(* CoDeSys 2.3 export: CELA.EXP *)

(* Data type in EPT Lib/Achsen/BECKHOFF *)
TYPE enum_ecd_cmd :
	(
	NO_COMMAND := 0,
	ABORT,
	POWER_DISABLE,
	POWER_ENABLE,
	RESET,
	HOME,
	SET_POSITION,
	JOG_VORWAERTS,
	JOG_RUECKWAERTS,
	JOG_STOP,
	MOVE_ABSOLUTE,
	MOVE_ABSOLUTE_NEXT,
	MOVE_RELATIVE,
	MOVE_VELOCITY,
	MOVE_MODULO,
	MOVE_TOUCH_PROBE,
	STOP_AXIS,
	HALT_AXIS,
	GEAR_IN_SLAVE,
	GEAR_OUT_SLAVE,
	CAM_IN_SLAVE,
	CAM_OUT_SLAVE,
	CAM_SCALEING_SLAVE,
	SOE_WRITE_PARAM,
	SOE_READ_PARAM,
	ECCOESDO_WRITE_PARAM,
	ECCOESDO_READ_PARAM,
	WRITE_NC_PARAMETER,
	READ_NC_PARAMETER,
	WRITE_ADS_PARAMETER,
	READ_ADS_PARAMETER,
	WRITE_MOTION_POINT,
	READ_MOTION_POINT,
	READ_SLAVE_DYNAMICS,
	READ_CAMTABLE_CHAR

	);
END_TYPE

(* Data type in EPT Lib/Achsen/BECKHOFF *)
TYPE enum_ecd_typ :
	(
	LINEAR := 1,
	RUND,
	LINEAR_VIRTUELL,
	RUND_VIRTUELL,
	SERVOKLEMME7201
	);
END_TYPE

(* Data type in EPT Lib/Achsen/BECKHOFF *)
TYPE st_camscaleingoptions :
STRUCT
	st_scaleing_activation_mode			: MC_CamActivationMode;
	r_scaleing_activation_position			: LREAL;
	st_master_scaling_mode				: MC_CamScalingMode;
	st_slave_scaling_mode				: MC_CamScalingMode;
END_STRUCT
END_TYPE

(* Data type in EPT Lib/Achsen/BECKHOFF *)
TYPE struct_achse :
STRUCT
	st_ctrl		: struct_ctrl;
	st_config		: struct_ecd_config;
	st_visu		: struct_ecd_visu;
END_STRUCT
END_TYPE

(* Data type in EPT Lib/Achsen/BECKHOFF *)
TYPE struct_ads_info :
STRUCT
	s_net_id 								: T_AmsNetId := '';
	st_symbol_info						: SYMINFOSTRUCT;
	dw_zieladresse_ads_read				: DWORD := 16#0000;
	dw_quelladresse_ads_write				: DWORD := 16#0000;
END_STRUCT
END_TYPE

(* Data type in EPT Lib/Achsen/BECKHOFF *)
TYPE struct_eccoe_sdo :
STRUCT
	s_ec_slave_net_id 		: T_AmsNetId := '';
	ui16_slave_addr 			: UINT := 0; (* Address of the slave device.*)
	i8_sub_index 				: BYTE := 0; (* CANopen Sdo subindex.*)
	w_index 					: WORD := 16#00; (* CANopen Sdo index.*)
	dw_p_source_buffer 		: DWORD := 16#0000; (* Contains the address of the buffer containing the data to be send. *)
	dw_p_destination_buffer	: DWORD := 16#0000; (* Contains the address of the buffer for the received data. *)
	ui32_buffer_length 			: UDINT := 0; (* Contains the max. number of bytes to be received. *)
	ui32_value 				: UDINT := 0; (* variable to be written to the CoE Object *)
	ui16_value 				: UINT := 0; (* variable to be written to the CoE Object *)
	byte_value 				: BYTE := 16#00; (* variable to be written to the CoE Object *)
	bool_value 				: BOOL := FALSE; (* variable to be written to the CoE Object *)
END_STRUCT
END_TYPE

(* Data type in EPT Lib/Achsen/BECKHOFF *)
TYPE struct_ecd_cmd :
STRUCT
	b_job_fehler 		: BOOL := FALSE;
	enu_cmd			: enum_ecd_cmd;
	meldungen		: struct_ecd_cmd_meldungen;
END_STRUCT
END_TYPE

(* Data type in EPT Lib/Achsen/BECKHOFF *)
TYPE struct_ecd_cmd_meldungen :
STRUCT
	sm_power_enable					: BOOL := FALSE;
	sm_power_disable				: BOOL := FALSE;
	sm_reset							: BOOL := FALSE;
	sm_home						: BOOL := FALSE;
	sm_setposition					: BOOL := FALSE;
	sm_jog_vorwaerts					: BOOL := FALSE;
	sm_jog_rueckwaerts				: BOOL := FALSE;
	sm_move_absolute				: BOOL := FALSE;
	sm_move_relative					: BOOL := FALSE;
	sm_move_velocity				: BOOL := FALSE;
	sm_move_modulo					: BOOL := FALSE;
	sm_stop_axis						: BOOL := FALSE;
	sm_halt_axis						: BOOL := FALSE;
	sm_gear_in_slave					: BOOL := FALSE;
	sm_gear_out_slave				: BOOL := FALSE;
	sm_cam_in_slave					: BOOL := FALSE;
	sm_cam_out_slave				: BOOL := FALSE;
	sm_cam_scaleing_slave			: BOOL := FALSE;
	sm_motion_command_timeout		: BOOL := FALSE;
	sm_camgear_command_timeout	: BOOL := FALSE;
	sm_achse_nicht_referenziert		: BOOL := FALSE;
	sm_limit_positiv_erreicht			: BOOL := FALSE;
	sm_limit_negativ_erreicht			: BOOL := FALSE;
	sm_write_soe_parameter			: BOOL := FALSE;
	sm_read_soe_parameter			: BOOL := FALSE;
	sm_write_nc_parameter			: BOOL := FALSE;
	sm_read_nc_parameter			: BOOL := FALSE;
	sm_write_motion_funktion_point		: BOOL := FALSE;
	sm_read_motion_funktion_point		: BOOL := FALSE;
	sm_read_camtable_slave_dynamics	: BOOL := FALSE;
	sm_read_camtable_charakteristik	: BOOL := FALSE;
	sm_write_ads_parameter			: BOOL := FALSE;
	sm_read_ads_parameter			: BOOL := FALSE;
	sm_ec_coe_sdo_write_ex			: BOOL := FALSE;
	sm_ec_coe_sdo_read_ex			: BOOL := FALSE;
	sm_touch_probe_defect			: BOOL := FALSE;
	sm_touch_probe_err				: BOOL := FALSE;
END_STRUCT
END_TYPE

(* Data type in EPT Lib/Achsen/BECKHOFF *)
TYPE struct_ecd_config :
STRUCT
	s_instanz_name					: STRING(48) := '';
	s_beschreibung					: STRING(32) := '';
	i16_meld_startindex				: INT;
	ui16_ethercat_adr					: UINT := 0;
	ui16_ethercat_slave_id				: UINT := 0;

	i16_achs_nr						: INT := 0;
	i16_modul_nr						: INT := 0;

	b_refsensor_vorhanden			: BOOL := FALSE;
	b_limitsensor_positiv_vorhanden	: BOOL := FALSE;
	b_limitsensor_negativ_vorhanden	: BOOL := FALSE;

	r_getriebefaktor					: LREAL := 0.0;
	ui16_bipolar_torque_limit			: UINT := 1000;
	i16_achstyp						: enum_ecd_typ;

	b_config_fertig					: BOOL := FALSE;
END_STRUCT
END_TYPE

(* Data type in EPT Lib/Achsen/BECKHOFF *)
TYPE struct_ecd_fehler :
STRUCT
	b_sammel				: BOOL := FALSE;
	b_job_fehler 				: BOOL := FALSE;
	b_achsfehler 				: BOOL := FALSE;
	b_devicefehler 			: BOOL := FALSE;
	b_limit_positiv_erreicht 		: BOOL := FALSE;
	b_limit_negativ_erreicht	: BOOL := FALSE;
END_STRUCT
END_TYPE

(* Data type in EPT Lib/Achsen/BECKHOFF *)
TYPE struct_ecd_geschwindigkeiten :
STRUCT
	lr_maximalgeschwindigkeit	: LREAL := 0.0;
	lr_beschleunigung 		: LREAL := 0.0;
	lr_verzoegerung	 		: LREAL := 0.0;
	lr_ruck			 		: LREAL := 0.0;

	lr_auto_max				: LREAL := 0.0;
	lr_auto_min				: LREAL := 0.0;
	lr_jog					: LREAL := 0.0;
END_STRUCT
END_TYPE

(* Data type in EPT Lib/Achsen/BECKHOFF *)
TYPE struct_ecd_meldungen :
STRUCT
	b_achsfehler					: BOOL := FALSE;
	b_devicefehler				: BOOL := FALSE;
	b_achse_nicht_bb				: BOOL := FALSE;
	b_achse_nicht_referenziert		: BOOL := FALSE;
	b_keine_verfahrfreigabe		: BOOL := FALSE;
	b_achse_nicht_auf_startpos		: BOOL := FALSE;
	b_ende_skalierungs_nocke		: BOOL := FALSE;
	b_ende_camming_nocke		: BOOL := FALSE;
	b_skalierung_noch_aktiv		: BOOL := FALSE;
END_STRUCT
END_TYPE

(* Data type in EPT Lib/Achsen/BECKHOFF *)
TYPE struct_ecd_positionen :
STRUCT
	r_soll		 			: LREAL := 0.0;
	r_referenz				: LREAL := 0.0;
	lr_ibn_pos_start			: LREAL := 0.0;
	lr_ibn_pos_ziel			: LREAL := 0.0;
END_STRUCT
END_TYPE

(* Data type in EPT Lib/Achsen/BECKHOFF *)
TYPE struct_ecd_visu :
STRUCT
	b_nullpunkt_setzen				: BOOL := FALSE;
	b_tippen_vorwaerts				: BOOL := FALSE;
	b_tippen_rueckwaerts				: BOOL := FALSE;
	b_achse_lueften					: BOOL := FALSE;
	b_achse_regeln					: BOOL := FALSE;
	b_bandeinzug_referenzieren		: BOOL := FALSE;
	i32_geschwindigkeit_soll			: DINT := 0;
	i32_geschwindigkeit_ist			: DINT := 0;
	i32_position_ist					: DINT := 0;
	lr_geschwindigkeit_soll				: LREAL := 0.0;
	lr_geschwindigkeit_ist				: LREAL := 0.0;
	lr_position_ist						: LREAL := 0.0;
	b_winkel_vor_ot_uebernehmen		: BOOL := FALSE;
	b_winkel_nach_ot_uebernehmen	: BOOL := FALSE;
	b_winkeloffset_uebernehmen		: BOOL := FALSE;
	b_einschalten						: BOOL := FALSE;
	b_ausschalten					: BOOL := FALSE;
	b_motor_dreht					: BOOL := FALSE;
	b_taste_vorgabegeschwindigkeit	: BOOL := FALSE;
	b_taste_plus						: BOOL := FALSE;
	b_taste_plusplus					: BOOL := FALSE;
	b_taste_minus					: BOOL := FALSE;
	b_taste_minusminus				: BOOL := FALSE;
	st_zyl							: struct_zylinder_visu;
END_STRUCT
END_TYPE

(* Data type in EPT Lib/Achsen/BECKHOFF *)
TYPE struct_nc_scaling_parameter :
STRUCT
	lr_ref_velo					: LREAL := 0.0;
	lr_max_velo					: LREAL := 0.0;
	lr_manual_velo_fast			: LREAL := 0.0;
	lr_manual_velo_slow			: LREAL := 0.0;
	lr_calibration_velo_forward		: LREAL := 0.0;
	lr_calibration_velo_backward	: LREAL := 0.0;
	lr_acceleration				: LREAL := 0.0;
	lr_deceleration				: LREAL := 0.0;
	lr_jerk						: LREAL := 0.0;
	lr_scaling_factor				: LREAL := 0.0;
END_STRUCT
END_TYPE

(* Data type in EPT Lib/Allgemeine Kontrollstrukturen Objekte *)
TYPE enum_step_nr :
	(
	INIT_OBJ := 0,
	INIT := 10,
	BEREIT := 100,
	FEHLER := 1000,
	STOP := 1100,
	STILLSTAND := 1200,
	HALT := 1300,
	HANDRAD := 2000,
	MOTORBREMSE_AUF :=2100,
	MOTORBREMSE_ZU := 2200,
	LUEFTEN := 2300,
	REGELN := 2400,
	NULLPUNKT_SETZEN := 2500,
	INBETRIEBNAHME := 5000,
	(* Zylinder *)
	ZYL_INIT := 3000,
	GESTOPPT := 3010,
	EINGEFAHREN := 3020,
	BEWEGUNG_AUSFAHREN := 3030,
	AUSGEFAHREN := 3040,
	BEWEGUNG_EINFAHREN := 3050,
	MITTEGEFAHREN := 3060,
	BEWEGUNG_MITTE := 3070,
	LUFTLOS := 3080,
	ZYL_FEHLER := 3090,
	DIREKT_EINFAHREN := 3100,
	DIREKT_AUSFAHREN := 3110
	);
END_TYPE

(* Data type in EPT Lib/Allgemeine Kontrollstrukturen Objekte *)
TYPE struct_config :
STRUCT
	str_instanz_name					: STRING(48) := '';
	str_beschreibung					: STRING(32) := '';
	b_station_aktiv					: BOOL := FALSE;
	b_station_in_simulation				: BOOL := FALSE;
	i16_meld_startindex				: INT := 0;
	b_config_fertig					: BOOL := FALSE;
END_STRUCT
END_TYPE

(* Data type in EPT Lib/Allgemeine Kontrollstrukturen Objekte *)
TYPE struct_ctrl :
STRUCT
	in		: struct_ctrl_in;
	out		: struct_ctrl_out;
END_STRUCT
END_TYPE

(* Data type in EPT Lib/Allgemeine Kontrollstrukturen Objekte *)
TYPE struct_ctrl_in :
STRUCT
	b_quitt						: BOOL := FALSE;
	b_stop 						: BOOL := FALSE;
         b_halt		  	 			: BOOL := FALSE;
         b_definierter_halt  	 			: BOOL := FALSE;
	b_init 						: BOOL := FALSE;
	b_init_2 						: BOOL := FALSE;
         b_preinit                				: BOOL := FALSE;
	b_start						: BOOL := FALSE;
	b_start_2						: BOOL := FALSE;
	b_gutteil_produziert 			: BOOL := FALSE;
	b_schlechtteil_produziert 		: BOOL := FALSE;
	b_start_lesen					: BOOL := FALSE;
	b_start_schreiben				: BOOL := FALSE;
	b_schutzhaube_ab			: BOOL := FALSE;
	b_schutzhaube_auf			: BOOL := FALSE;
	b_nachtabschaltung			: BOOL := FALSE;
	b_gehe_step_ibn				: BOOL := FALSE;
	b_ibn_start					: BOOL := FALSE;
	b_freigabe					: BOOL := FALSE;
	b_bremse_auf				: BOOL := FALSE;
	b_bremse_zu					: BOOL := FALSE;
	b_home						: BOOL := FALSE;
	b_ausfaedeln_servo			: BOOL := FALSE;
	b_einfaedeln_servo			: BOOL := FALSE;
	b_startpos					: BOOL := FALSE;
END_STRUCT
END_TYPE

(* Data type in EPT Lib/Allgemeine Kontrollstrukturen Objekte *)
TYPE struct_ctrl_out :
STRUCT
	b_bereit 						: BOOL := FALSE;
	b_bereit_2					: BOOL := FALSE;
         b_prebereit               			: BOOL := FALSE;
	b_fehler 						: BOOL := FALSE;
	b_fertig						: BOOL := FALSE;
	b_fertig_2					: BOOL := FALSE;
	b_bandende					: BOOL := FALSE;
	b_kontroller_start				: BOOL := FALSE;
	b_gestoppt					: BOOL := FALSE;
	b_angehalten					: BOOL := FALSE;
	b_haube_oeffnen				: BOOL := FALSE;
	b_nachtabschaltung			: BOOL := FALSE;
	b_einzelfertigung				: BOOL := FALSE;
	b_busy						: BOOL := FALSE;
	b_bremse_geschlossen		: BOOL := FALSE;
	b_bremse_geoeffnet			: BOOL := FALSE;
	b_ausgefaedelt_servo			: BOOL := FALSE;
	b_servo_auf_einfaedelpos		: BOOL := FALSE;
END_STRUCT
END_TYPE

(* Data type in EPT Lib/Allgemeine Kontrollstrukturen Objekte *)
TYPE struct_objekt :
STRUCT
	st_config		: struct_config;
	st_ctrl		: struct_ctrl;
	st_visu		: struct_visu;
END_STRUCT
END_TYPE

(* Data type in EPT Lib/Analogkarte *)
TYPE struct_analog_in :
STRUCT
	e_b_status_underrange		: BOOL := FALSE;
	e_b_status_overrange			: BOOL := FALSE;
	e_by_status_limit1				: BYTE := 2#0;
	e_by_status_limit2				: BYTE := 2#0;
	e_b_status_error				: BOOL := FALSE;
	e_i16_value					: INT := 0;
END_STRUCT
END_TYPE

(* Data type in EPT Lib/Analogkarte *)
TYPE struct_analogin :
STRUCT
	fb			: ST_AnalogIn;
	st_ctrl		: struct_ctrl;
END_STRUCT
END_TYPE

(* Data type in EPT Lib/Analogkarte *)
TYPE struct_analogout :
STRUCT
	fb			: ST_AnalogOut;
	st_ctrl		: struct_ctrl;
END_STRUCT
END_TYPE

(* Data type in EPT Lib/Betriebsarten *)
TYPE enum_betriebsarten :
	(KEINE := 0,
	AUTO,
	TIPPEN,
	DUMMY,
	PSEUDO,
	HAND);
END_TYPE

(* Data type in EPT Lib/Betriebsarten *)
TYPE struct_betriebsarten :
STRUCT
	st_config					: struct_config;
	st_ctrl					: struct_ctrl;
END_STRUCT
END_TYPE

(* Data type in EPT Lib/CamEditor *)
TYPE enum_auftrag_cameditor :
	(
	MFP_KEIN_AUFTRAG := 0,
	MFP_LESEN,
	MFP_SCHREIBEN
	);
END_TYPE

(* Data type in EPT Lib/CamEditor *)
TYPE struct_cam_editor :
STRUCT
	fb					: ST_Kurvenscheibeneditor;
	st_config				: struct_config;
	st_ctrl				: struct_ctrl;
END_STRUCT
END_TYPE

(* Data type in EPT Lib/CamEditor *)
TYPE struct_cameditor_meldungen :
STRUCT
	schreibe_mfp 							: BOOL := FALSE;
	lese_mfp									: BOOL := FALSE;
	schreibe_camtable						: BOOL := FALSE;
	lese_camtable							: BOOL := FALSE;
	berechne_konstantfahrphase				: BOOL := FALSE;
	berechne_max_master_geschwindigkeit		: BOOL := FALSE;
	lesen_werte_mf_tab						: BOOL := FALSE;
	fehler_cam_in								: BOOL := FALSE;
END_STRUCT
END_TYPE

(* Data type in EPT Lib/CamEditor *)
TYPE struct_camtable_maker :
STRUCT
	fb					: ST_Camtable_Maker;
	st_config			: struct_config;
	st_ctrl				: struct_ctrl;
END_STRUCT
END_TYPE

(* Data type in EPT Lib/CamEditor *)
TYPE struct_db_motionfunctionpoint :
STRUCT
	    PointIndex        		: MC_MotionFunctionPoint_ID;
	    FunctionType    		: MC_MotionFunctionType;
	    PointType        		: MC_MotionPointType;
	    MasterPos        		: LREAL; (* X *)
	    SlavePos          		: LREAL; (* Y *)
END_STRUCT
END_TYPE

(* Data type in EPT Lib/CamEditor *)
TYPE struct_mf_editor :
STRUCT
	fb					: ST_MFCalcConstPhase;
	st_config				: struct_config;
	st_ctrl				: struct_ctrl;
END_STRUCT
END_TYPE

(* Data type in EPT Lib/Diagnose *)
TYPE struct_ecat_klemmen_diagnose :
STRUCT
	WcState			: BOOL := 2#0;		(* 1 = Data invalid *)
	ECatState		: UINT := 0;		(* 0x08 = OP-State *)
END_STRUCT
END_TYPE

(* Data type in EPT Lib/Nockenschaltwerk/NSW_INT *)
TYPE struct_nocken_int :
STRUCT
	i16_track_no 				: INT := 0;
	b_camvalid 				: BOOL := FALSE;
	b_eff_direction_pos 		: BOOL := FALSE;
	b_eff_direction_neg 		: BOOL := FALSE;
	b_nockenzustand 			: BOOL := FALSE;
	i16_cam_begin 			: INT := 0;
	i16_cam_end 				: INT := 0;
	t_vorsteuerzeit			: TIME := t#0ms;
	i16_vorsteuerpos			: INT := 0;
END_STRUCT
END_TYPE

(* Data type in EPT Lib/Nockenschaltwerk/NSW_INT *)
TYPE struct_nockenschaltwerk_int :
STRUCT
	fb					: ST_Nockenschaltwerk_int;
	st_config				: struct_config;
	arr_nocken			: ARRAY [0..MAX_NOCKENGERUEST] OF struct_nocken_int;
	arr_spur				: ARRAY [0..MAX_NOCKENGERUEST] OF BOOL;
END_STRUCT
END_TYPE

(* Data type in EPT Lib/Nockenschaltwerk/NSW_LREAL *)
TYPE struct_nocken_lreal :
STRUCT
	i16_track_no 				: INT := 0;
	b_camvalid 				: BOOL := FALSE;
	b_eff_direction_pos 		: BOOL := FALSE;
	b_eff_direction_neg 		: BOOL := FALSE;
	b_nockenzustand 			: BOOL := FALSE;
	r_cam_begin 				: LREAL := 0.0;
	r_cam_end 				: LREAL := 0.0;
	t_vorsteuerzeit			: TIME := t#0ms;
	r_vorsteuerpos			: LREAL := 0.0;
END_STRUCT
END_TYPE

(* Data type in EPT Lib/Nockenschaltwerk/NSW_LREAL *)
TYPE struct_nocken_visu :
STRUCT
	b_daten_backup					: BOOL := FALSE;
	b_daten_recover					: BOOL := FALSE;
	b_setze_drehgeber_nullpunkt		: BOOL := FALSE;
END_STRUCT
END_TYPE

(* Data type in EPT Lib/Nockenschaltwerk/NSW_LREAL *)
TYPE struct_nockeneinstellungen :
STRUCT
	arr_nocken			: ARRAY [0..MAX_NOCKENGERUEST] OF struct_nocken_lreal;
END_STRUCT
END_TYPE

(* Data type in EPT Lib/Nockenschaltwerk/NSW_LREAL *)
TYPE struct_nockenschaltwerk_lreal :
STRUCT
	fb					: ST_Nockenschaltwerk_lreal;
	st_config				: struct_config;
	arr_nocken			: ARRAY [0..MAX_NOCKENGERUEST] OF struct_nocken_lreal;
	arr_spur				: ARRAY [0..MAX_NOCKENGERUEST] OF BOOL;
END_STRUCT
END_TYPE

(* Data type in EPT Lib/Nockenschaltwerk/NZW *)
TYPE struct_nockenzaehlwerk :
STRUCT
	fb					: ST_Nockenzaehlwerk;
	st_config				: struct_config;
END_STRUCT
END_TYPE

(* Data type in EPT Lib/Routing *)
TYPE struct_ads_kommunikation :
STRUCT
	fb			: ST_ADS_Kommunikation;
END_STRUCT
END_TYPE

(* Data type in EPT Lib/Routing *)
TYPE struct_nachbar_pc :
STRUCT
	st_station_vorher		: struct_station_vorher;
	st_station_nachher		: struct_station_nachher;
END_STRUCT
END_TYPE

(* Data type in EPT Lib/Routing *)
TYPE struct_station_nachher :
STRUCT
	s_ams_netid		: T_AmsNetId := '0.0.0.0.0.0';
	in				: struct_station_nachher_in;
	out				: struct_station_nachher_out;
END_STRUCT
END_TYPE

(* Data type in EPT Lib/Routing *)
TYPE struct_station_nachher_in :
STRUCT
	b_erlaubnis			: BOOL;
	b_angekommen		: BOOL;
END_STRUCT
END_TYPE

(* Data type in EPT Lib/Routing *)
TYPE struct_station_nachher_out :
STRUCT
	b_start_fb			: BOOL;
END_STRUCT
END_TYPE

(* Data type in EPT Lib/Routing *)
TYPE struct_station_vorher :
STRUCT
	s_ams_netid		: T_AmsNetId := '0.0.0.0.0.0';
	in				: struct_station_vorher_in;
	out				: struct_station_vorher_out;
END_STRUCT
END_TYPE

(* Data type in EPT Lib/Routing *)
TYPE struct_station_vorher_in :
STRUCT
	b_start_fb			: BOOL;
END_STRUCT
END_TYPE

(* Data type in EPT Lib/Routing *)
TYPE struct_station_vorher_out :
STRUCT
	b_erlaubnis			: BOOL;
	b_angekommen		: BOOL;
END_STRUCT
END_TYPE

(* Data type in EPT Lib/Serielle Kommunikation *)
TYPE struct_balluff_tag_reader :
STRUCT
	fb			: ST_BalluffTagReader;
	st_ctrl		: struct_ctrl;
END_STRUCT
END_TYPE

(* Data type in EPT Lib/Serielle Kommunikation *)
TYPE struct_barcode_reader :
STRUCT
	fb			: ST_BarcodeReader;
	st_ctrl		: struct_ctrl;
END_STRUCT
END_TYPE

(* Data type in EPT Lib/Serielle Kommunikation *)
TYPE struct_serial_data :
STRUCT
	arr_buffer			: ARRAY[0..79] OF BYTE;
	i32_size				: UDINT := 0;
END_STRUCT
END_TYPE

(* Data type in EPT Lib/Sprache *)
TYPE enum_sprache :
	(
	KEINE_SPRACHE := 0,
	DEUTSCH := 1,
	ENGLISCH := 2,
	TSCHECHISCH := 3,
	RESERVESPRACHE1 := 4,
	RESERVESPRACHE2 := 5);
END_TYPE

(* Data type in EPT Lib/Sprache *)
TYPE struct_sprachumschaltung :
STRUCT
	i16_akt_sprache		: enum_sprache := DEUTSCH;
END_STRUCT
END_TYPE

(* Data type in EPT Lib/Zylinder *)
TYPE struct_st_zylinder :
STRUCT
	fb			: ST_Zylinder12V012346E;
	st_ctrl		: struct_zylinder_ctrl;
END_STRUCT
END_TYPE

(* Data type in EPT Lib/Zylinder *)
TYPE struct_totzeitkompensation :
STRUCT
	t_einfahrzeit					: TIME := t#0ms;
	t_ausfahrzeit					: TIME := t#0ms;
	t_einfahrzeit_kompensiert		: TIME := t#0ms;
	t_ausfahrzeit_kompensiert		: TIME := t#0ms;
	t_kompensationszeit			: TIME := t#0ms;
	fb_ton_tzk					: TON;
END_STRUCT
END_TYPE

(* Data type in EPT Lib/Zylinder *)
TYPE struct_zylinder_config :
STRUCT
	i16_identnummer					: INT := 0;
	i16_gruppe						: INT := 0;
	str_instanz_name					: STRING(48) := '';
	str_beschreibung					: STRING(32) := '';
	str_zylinder_typ					: STRING := '2V2E_EIN_AUS';
	b_aktiv							: BOOL := TRUE;
	b_endlage1_aktiv					: BOOL := TRUE;
	b_sensor1_aktiv					: BOOL := TRUE;
	b_endlage2_aktiv	 				: BOOL := FALSE;
	b_sensor2_aktiv					: BOOL := FALSE;
	b_endlage3_aktiv	 				: BOOL := FALSE;
	b_sensor3_aktiv					: BOOL := FALSE;
	t_ueberwachungszeit				: TIME := t#2000ms;
	t_ein_aus_fahrzeit					: TIME := t#100ms;
	i16_meld_startindex				: INT := 0;
	i16_tzk_faktor_ausfahren			: INT := 100;
	i16_tzk_faktor_einfahren			: INT := 100;
	b_config_fertig					: BOOL := FALSE;
END_STRUCT
END_TYPE

(* Data type in EPT Lib/Zylinder *)
TYPE struct_zylinder_ctrl :
STRUCT
	in		: struct_zylinder_ctrl_in;
	out		: struct_zylinder_ctrl_out;
END_STRUCT
END_TYPE

(* Data type in EPT Lib/Zylinder *)
TYPE struct_zylinder_ctrl_in :
STRUCT
	b_quittieren			: BOOL := FALSE;
	b_stop				: BOOL := FALSE;
	b_einfahren			: BOOL := FALSE;
	b_ausfahren			: BOOL := FALSE;
	b_luftlos				: BOOL := FALSE;
END_STRUCT
END_TYPE

(* Data type in EPT Lib/Zylinder *)
TYPE struct_zylinder_ctrl_out :
STRUCT
	b_fehler				: BOOL := FALSE;
	b_eingefahren		: BOOL := FALSE;
	b_ausgefahren		: BOOL := FALSE;
	b_gestoppt			: BOOL := FALSE;
	b_ohne_luft			: BOOL := FALSE;
END_STRUCT
END_TYPE

(* Data type in EPT Lib/Zylinder *)
TYPE struct_zylinder_meldungen :
STRUCT
	b_zeit_ausfahren1			: BOOL := FALSE;
	b_zeit_einfahren1			: BOOL := FALSE;
	b_endlage1				: BOOL := FALSE;
	b_sensor1				: BOOL := FALSE;
	b_zeit_ausfahren2			: BOOL := FALSE;
	b_zeit_einfahren2			: BOOL := FALSE;
	b_endlage2				: BOOL := FALSE;
	b_sensor2				: BOOL := FALSE;
	b_zeit_ausfahren3			: BOOL := FALSE;
	b_zeit_einfahren3			: BOOL := FALSE;
	b_endlage3				: BOOL := FALSE;
	b_sensor3				: BOOL := FALSE;
	b_winkel_ausfahren1		: BOOL := FALSE;
	b_winkel_einfahren1		: BOOL := FALSE;
	b_winkel_ausfahren2		: BOOL := FALSE;
	b_winkel_einfahren2		: BOOL := FALSE;
	b_winkel_ausfahren3		: BOOL := FALSE;
	b_winkel_einfahren3		: BOOL := FALSE;
	b_zyltyp_nicht_definiert		: BOOL := FALSE;
	b_reserve1				: BOOL := FALSE;
END_STRUCT
END_TYPE

(* Data type in EPT Lib/Zylinder *)
TYPE struct_zylinder_visu :
STRUCT
	b_taste_ausfahren			: BOOL := FALSE;
	b_taste_mittefahren		: BOOL := FALSE;
	b_taste_einfahren			: BOOL := FALSE;
	b_sensor_eingefahren		: BOOL := FALSE;
	b_sensor_ausgefahren		: BOOL := FALSE;
	b_sensor_mittegefahren	: BOOL := FALSE;
	enu_zustand				: enum_step_nr;
	i16_nr_zyl_im_handbetrieb	: INT := 0;
	i16_zyl_id 				: INT := 0;
	i16_zyl_fehlergruppe		: INT := 0;
END_STRUCT
END_TYPE

(* Data type in Gemeinsamkeiten17xx/Allgemein *)
TYPE enum_achsen :
	(
	KEINE_ACHSE := 0,
	BESTUECK__ACHSE := 1,
	Z__ACHSE := 2,
	Y__ACHSE := 3,
	B__ACHSE := 4);
END_TYPE

(* Data type in Gemeinsamkeiten17xx/Allgemein *)
TYPE enum_maschinenstatus :
	(
	KEIN_STATUS := 0,
	STATUS_FEHLER := 1,
	STATUS_FEHLER_QUITTIERT := 2,
	STATUS_BETRIEBSBEREIT := 3,
	STATUS_MASCHINE_ARBEITET := 4);
END_TYPE

(* Data type in Gemeinsamkeiten17xx/Allgemein *)
TYPE enum_raster :
	(
	KEIN_RASTER := 0,
	RASTER_DEFAULT,
	RASTER_22,
	RASTER_34);
END_TYPE

(* Data type in Gemeinsamkeiten17xx/Allgemein *)
TYPE enum_typ_Bestueckprog :
	(
	BESTUECKUNG_AUTO := 0,
	BESTUECKUNG_HALBAUTO:=1,
	BESTUECKUNG_MANUAL:=5
	);
END_TYPE

(* Data type in Gemeinsamkeiten17xx/Allgemein *)
TYPE enum_typ_zelle :
	(
	KEINE_ZELLE := 0,
	BESTUECKZELLE_1700,
	BESTUECKZELLE_1720,
	RASTERFOLIE
	);
END_TYPE

(* Data type in Gemeinsamkeiten17xx/Barcode *)
TYPE struct_barcode :
STRUCT
	fb			: ST_Barcode;
END_STRUCT
END_TYPE

(* Data type in Gemeinsamkeiten17xx/Barcode *)
TYPE struct_barcode_daten :
STRUCT
	(* Angewählte Bänder und Wkz *)
	s_wkz_anwahl				: STRING;
	s_band_anwahl				: STRING;
	s_band_ID_links				: STRING:='';
	s_band_ID_rechts			: STRING:='';

	(* Dürfen diese Bander verarbeitet werden ?*)
	b_band_links_ok				: BOOL;
	b_band_rechts_ok				: BOOL;
	b_band_ok					: BOOL;
	b_band_ID_links_ok				: BOOL;
	b_band_ID_rechts_ok				: BOOL;
END_STRUCT
END_TYPE

(* Data type in Gemeinsamkeiten17xx/BBGen/PersDaten *)
TYPE struct_LTS :
STRUCT
	s_tmpNewbatch				: ARRAY [0..1] OF STRING(20);
	i_tmpVPE					: DINT;

END_STRUCT
END_TYPE

(* Data type in Gemeinsamkeiten17xx/BBGen/PersDaten *)
TYPE struct_LTS_xml :
STRUCT
	timestamp					: STRING(20);	(*Zeitstempel*)
	order						: STRING(20);	(*(Fertigungsaftrag) wird nur an der UML beschrieben muss aber in der xml Struktur vorhanden sein *)
	newbatch					: ARRAY [0..1] OF STRING(20);	(*Chargennummer (ID)  ARRAY 1 wid nur bei 1720 benutzt*)
	VPE						: DINT;			(*Verpackungseinheit*)
	UmlNo						: DINT;			(*Anlagennummer UML kommt mit der Plle mit*)
END_STRUCT
END_TYPE

(* Data type in Gemeinsamkeiten17xx/BBGen/PersDaten *)
TYPE struct_PD :
STRUCT
	st_LTS						: struct_LTS;

	b_Zelle_nicht_in_Betrieb		: BOOL;
	i_DayOfYearAutoCheckIn	: DINT;

END_STRUCT
END_TYPE

(* Data type in Gemeinsamkeiten17xx/BBGen *)
TYPE enum_bandtyp :
(
	ZINN := 0,
	GOLD,
	SILBER
);
END_TYPE

(* Data type in Gemeinsamkeiten17xx/BBGen *)
TYPE enum_bbgen_auftrag :
(
	KEIN_BB_AUFTRAG := 0,
	LESE_WKZ,
	LESE_MD,
	LESE_ISK,
	LESE_BAND,
	LESE_WT,
	LESE_BESTUECKBILD,
	LESE_KOMPLETT,
	SCHREIBE_ISK,
	SCHREIBE_WKZ,
	SCHREIBE_BAND,
	SCHREIBE_WT,
	SCHREIBE_MD,
	SCHREIBE_BESTUECKBILD
);
END_TYPE

(* Data type in Gemeinsamkeiten17xx/BBGen *)
TYPE enum_bestueckrichtung :
(
	YMinus_nach_YPlus_ZMinus_nach_ZPlus := 0,
	YMinus_nach_YPlus_ZPlus_nach_ZMinus,
	YPlus_nach_YMinus_ZMinus_nach_ZPlus,
	YPlus_nach_YMinus_ZPlus_nach_ZMinus
);
END_TYPE

(* Data type in Gemeinsamkeiten17xx/BBGen *)
TYPE enum_typ_bandeinzug :
(
	KEIN_EINZUG := 0,
	STANDARD_2FACH_V2:=2,
	BANDWECHSLER_V2:=4,
	SERVO:=5
);
END_TYPE

(* Data type in Gemeinsamkeiten17xx/BBGen *)
TYPE enum_typ_bandeinzug_visu :
(
	KEIN_BANDEINZUG := 0,
	BANDEINZUG_1,
	BANDEINZUG_2,
	BANDEINZUG_3
);
END_TYPE

(* Data type in Gemeinsamkeiten17xx/BBGen *)
TYPE enum_typ_wkz :
(
	NORMAL := 0,
	BESTUECKSCHIEBER_GESTEUERT:=1
);
END_TYPE

(* Data type in Gemeinsamkeiten17xx/BBGen *)
TYPE struct_banddaten :
STRUCT
	typ					: enum_bandtyp;
	st_einpressen		: struct_einpresskraftueberwachung;
	r_raster				: LREAL := 0.0;
	i16_igelrad_zaehne	: INT := 0;
	i16_startpos_einfaedeln : INT := 0;
	lr_offset_erster_hub_wkz_mm	: LREAL := 0.0;
END_STRUCT
END_TYPE

(* Data type in Gemeinsamkeiten17xx/BBGen *)
TYPE struct_bestueckbild :
	(* Struktur beschreibt einen kompletten Stecker mit allen Daten *)
STRUCT
	(* Artikel *)
	s_artikelnummer			: STRING(50);
	(* Beschreibung des Projekts *)
	s_beschreibung			: STRING(50);

	(* Werkzeug Wechselteil(WT) *)
	s_wkzgruppe				: ARRAY [0..4] OF struct_wkzgruppe;

	(* Der zu verarbeitende ISK *)
	s_isknummer				: STRING(50);
	(* Projektnummer *)
	s_projektnummer			: ARRAY  [0..4] OF STRING(4);

	(* Bestückrichtung *)
	enu_richtung			 	: enum_bestueckrichtung;

	(* Alle Pins innerhalb dieses Steckers *)
	i32_anzahl_pins			: DINT := 0;
	s_Bestueckbild_vollbestueckt	: ARRAY  [0..14] OF STRING(255);
	st_pins					: ARRAY  [0..1023] OF struct_PinDaten;

END_STRUCT
END_TYPE

(* Data type in Gemeinsamkeiten17xx/BBGen *)
TYPE struct_bestueckbild_halbauto :
	(* Struktur beschreibt einen kompletten Stecker mit allen Daten *)
STRUCT
	(* bei TRUE liest der UML Desinger das Bestückbild nicht ein *)
	b_uml_designer_ignore	: BOOL := FALSE;
	(* Artikel *)
	s_artikelnummer			: STRING(50);
	(* Beschreibung des Projekts *)
	s_beschreibung			: STRING(50);

	(* Werkzeug Wechselteil(WT) *)
	s_wkzgruppe				: ARRAY [0..4] OF struct_wkzgruppe;

	(* Der zu verarbeitende ISK *)
	s_isknummer				: STRING(50);
	(* Projektnummer *)
	s_projektnummer			: ARRAY  [0..4] OF STRING(4);

	st_uml_designer_isk			: ARRAY [0..7] OF struct_uml_designer_isk;

	s_Bestueckbild_vollbestueckt	: ARRAY  [0..14] OF STRING(255);

	Wkz							:ARRAY  [0..14] OF struct_bestueckprogramm;

END_STRUCT
END_TYPE

(* Data type in Gemeinsamkeiten17xx/BBGen *)
TYPE struct_bestueckprogramm :
STRUCT

	i32_anzahl						: DINT := 0;
	s_band							: STRING(20);
	lr_y_offset						: LREAL;
	lr_z_offset						: LREAL;
	st_isk							: struct_isk_daten;
	lr_y								: ARRAY [0..511] OF LREAL;
	lr_z								: ARRAY [0..511] OF LREAL;
	i16_b							: ARRAY [0..511] OF INT;
	b_podest_verschieben			: ARRAY [0..511] OF BOOL;
END_STRUCT
END_TYPE

(* Data type in Gemeinsamkeiten17xx/BBGen *)
TYPE struct_datensatz :
STRUCT
	st_bestueckprogramm					: struct_bestueckprogramm;
	st_isk								: struct_isk_daten;
	st_band								: struct_banddaten;
	st_wkz								: struct_wkz;
	st_wt								: struct_wt;
	st_md								: struct_maschinendaten;
	st_stueckzahlen						: struct_stueckzahlen;
	st_wartungsprotokoll					: struct_Wartungsprotokoll;


	i16_counter_pruef_pos1				: DINT;
	i16_counter_pruef_pos2				: DINT;

END_STRUCT
END_TYPE

(* Data type in Gemeinsamkeiten17xx/BBGen *)
TYPE struct_isk_daten :
STRUCT
	lr_breite		: LREAL;
	lr_hoehe		: LREAL;
	lr_pos_y_0	: LREAL;
	lr_pos_z_0	: LREAL;
END_STRUCT
END_TYPE

(* Data type in Gemeinsamkeiten17xx/BBGen *)
TYPE struct_maschinendaten :
STRUCT
	i16_typ_zelle						: enum_typ_zelle := KEINE_ZELLE;
	i16_typ_y_achse					: INT;
	i32_bestueckhubzaehler				: UDINT := 0;
	T_Betriebstundenzaehler_alt			:TIME;
	T_Betriebstundenzaehler_neu		:TIME;

	(* Bestückbildgenerierung: speichern der aktuellen Daten, welche für den Neustart der Maschine notwendig sind. *)
	s_aktuelles_wkz						: STRING(50);
	s_aktuelles_wkz_wartung			: STRING(50);
	s_aktuelles_band					: STRING(50);
	s_aktuelle_artikelnummer				: STRING(50);
	s_aktueller_isk						: STRING(50);
	s_aktueller_wt						: STRING(50);

	b_wt_transport_aktiv					: BOOL := FALSE;
	b_hublift_links_aktiv					: BOOL := FALSE;
	b_hublift_rechts_aktiv				: BOOL := FALSE;
	b_wt_transport_simulation			: BOOL := FALSE;
	b_hublift_links_simulation				: BOOL := FALSE;
	b_hublift_rechts_simulation			: BOOL := FALSE;
	b_auto_Bandwechsel				: BOOL := FALSE;

	st_md_bestueckachse				: struct_md_achse;
	st_md_z_achse						: struct_md_achse;
	st_md_y_achse						: struct_md_achse;
	st_md_b_achse						: struct_md_achse;
	st_md_transport_wt_achse			: struct_md_achse;

	st_rasterplatte						: struct_daten_rasterplatte;

	b_bestueckprogramm_manuell		: BOOL := FALSE;	(* Haken wird in Visu gesetzt *)
	i16_typ_bestueckmodus				: enum_typ_Bestueckprog := BESTUECKUNG_AUTO;
	b_tagreader_fahrend					: BOOL := FALSE;

	i32_betriebssekundenzaehler			: UDINT := 0;
	i16_tag_data_structur_version		: INT := 0; (* 0 =Version mit StateParts[0]/[1], 1 = Version mit StateParts[0..7] *)
	i32_werkzeughubzaehler				: UDINT := 0;
	b_band_ID_Puffer_aus				: BOOL := FALSE;
	b_haspel_mit_auflegeblech			: BOOL := FALSE;	(*Wird im Programm nicht mehr verwendet, weil alle Zellen nachgerüstet wurden*)
	lr_offset_z_pos_0					: LREAL := 0.0;
	lr_offset_y_pos_0					: LREAL := 0.0;
	st_wkz_gruppe						: ARRAY[0..4] OF  struct_md_wkz; (*nur bei Halbautomatisch: Werkzeuge die mann zusammenfassen kann*)
	lr_ToleranzTouchProbe				: LREAL := 0.1;
	i16_WdhTouchProbe				: INT := 0;
	t_max_Traegerwechselzeit			:TIME:=t#1200ms;
	t_max_Tischwechselzeit			:TIME:=t#500ms;
	produzierte_Stecker				: UDINT;
	b_auswahlSpruehoeler				: BOOL:=TRUE;
	b_wkzBereinigen					:BOOL:=FALSE;		(*wenn true dann wird die Werkzeugdatei vorher gelöscht und dann neu erstellt*)
	r_geschwindigkeit_achse_transport		: LREAL := 0.0;
	b_anwahl_transport_achse			: BOOL := FALSE;	(* wenn TRUE, dann ist Transport-Achse für schnellen WT-Wechsel vorhanden *)
END_STRUCT
END_TYPE

(* Data type in Gemeinsamkeiten17xx/BBGen *)
TYPE struct_md_achse :
STRUCT
	lr_startposition						: LREAL;
	lr_nullpunktverschiebung				: LREAL;
	lr_wt_uebergabepos					: LREAL;
END_STRUCT
END_TYPE

(* Data type in Gemeinsamkeiten17xx/BBGen *)
TYPE struct_md_wkz :
STRUCT
	s_wkz						: STRING(50);
	i16_wkz_gruppe_kompatibel	: INT;
	s_Band						: STRING(50);
	i32_Anzahl					: DINT;
	i32_Wkz_nr					: DINT;
END_STRUCT
END_TYPE

(* Data type in Gemeinsamkeiten17xx/BBGen *)
TYPE struct_pindaten :
STRUCT
	lr_y	:	LREAL;
	lr_z	:	LREAL;
	typ	:	STRING(50);
END_STRUCT
END_TYPE

(* Data type in Gemeinsamkeiten17xx/BBGen *)
TYPE struct_uml_designer_isk :
STRUCT
	s_isknummer		: STRING(20);
	lr_y_offeset			: LREAL := 0.0;
	lr_z_offeset			: LREAL := 0.0;
END_STRUCT
END_TYPE

(* Data type in Gemeinsamkeiten17xx/BBGen *)
TYPE struct_virtmaster_bestueckachse :
STRUCT
	arr_motion_function_points	: ARRAY[1..100] OF struct_db_motionfunctionpoint;
END_STRUCT
END_TYPE

(* Data type in Gemeinsamkeiten17xx/BBGen *)
TYPE struct_wkz :
STRUCT
	i16_anzahl_einfaedel_pins				: INT := 1;
	i16_anzahl_einfaedel_auto_pins			: INT := 1;
	b_laufrichtung_haspel_links				: BOOL := FALSE;
	b_wkz_blasluft_aktiv					: BOOL := FALSE;
	nockenschaltwerk_bestueckachse		: struct_nockeneinstellungen;

	b_wkz_zweifachfallend					: BOOL := FALSE;
	r_auto								: LREAL := 0.0;
	r_auto_y								: LREAL := 0.0;
	r_auto_z								: LREAL := 0.0;
	r_auto_bandeinzug					: LREAL := 0.0;
	st_yz_tisch							: struct_yz_tisch;
	lr_offset_z_pos_0						: LREAL := 0.0;
	lr_offset_y_pos_0						: LREAL := 0.0;

	st_rasterfolie							: struct_daten_rasterfolie;

	i16_typ_bandeinzug					: enum_typ_bandeinzug := KEIN_EINZUG;

	st_oeler								: struct_oeler;

	lr_einfaedelposition					: LREAL := 180.0;
	i16_typ_wkz							: enum_typ_wkz := NORMAL;
	i16_anzahl_bestueckschieber			: INT := 1;
	i16_wkz_gruppe_kompatibel			: INT; 		(*Werkzeuge die die Gleiche Arbeit machen können sollten die gleiche Nummer haben*)

	b_rafo_vorzentrierer_aktiv				: BOOL := FALSE;
	i16_einfaedelhub_lueften				: INT := 1;
	b_variable_einfahrposition				: BOOL := FALSE;
	i16_anzahl_Teile_autostop_bandwechsel	: INT := 0;
	lr_ausbauposition						: LREAL := 17.0;
	i16_vorgabe_einfaedeln					: INT := 3;
	b_rafo_auto_einf_aktiv					: BOOL := FALSE;
	bFahreSofortAufUebergabePosition		: BOOL := FALSE;
END_STRUCT
END_TYPE

(* Data type in Gemeinsamkeiten17xx/BBGen *)
TYPE struct_wkzgruppe :
STRUCT
	s_wkznummer			: ARRAY [0..MaxNoOfWkz] OF STRING(50);
END_STRUCT
END_TYPE

(* Data type in Gemeinsamkeiten17xx/BBGen *)
TYPE struct_wt :
STRUCT
	lr_offset_z_pos_0						: LREAL := 0.0;
	lr_offset_y_pos_0						: LREAL := 0.0;
	i_anzahl_teile							: INT := 1;
	i16_typ_bestueckmodus				: enum_typ_Bestueckprog := BESTUECKUNG_AUTO;
END_STRUCT
END_TYPE

(* Data type in Gemeinsamkeiten17xx/BBGen *)
TYPE struct_yz_tisch :
STRUCT
	r_wkz_einfahrpos_z		: LREAL := 0.0;
	r_wkz_einfahrpos_y		: LREAL := 0.0;
END_STRUCT
END_TYPE

(* Data type in Gemeinsamkeiten17xx/Betriebsfreigaben *)
TYPE struct_betriebsfreigaben :
STRUCT
	st_config		: struct_config;
	st_ctrl		: struct_ctrl;
END_STRUCT
END_TYPE

(* Data type in Gemeinsamkeiten17xx/Betriebsstundenzaehler *)
TYPE struct_betriebsstundenzaehler :
STRUCT
	fb			: ST_Betriebsstundenzaehler;
	st_ctrl		: struct_ctrl;
END_STRUCT
END_TYPE

(* Data type in Gemeinsamkeiten17xx/Haspel *)
TYPE struct_einfach_haspelkontroller :
STRUCT
	fb			: ST_Einfachhaspelkontroller;
	st_ctrl		: struct_ctrl;
	st_visu		: struct_visu;
END_STRUCT
END_TYPE

(* Data type in Gemeinsamkeiten17xx/Haspel *)
TYPE struct_haspel_st_zylinder :
STRUCT
	fb			: ST_Haspel_st_zylinder;
	st_ctrl		: struct_ctrl;
	st_visu		: struct_visu;
END_STRUCT
END_TYPE

(* Data type in Gemeinsamkeiten17xx/Haspel *)
TYPE struct_haspel_V2 :
STRUCT
	fb			: ST_Haspel_V2;
	st_ctrl		: struct_ctrl;
	st_visu		: struct_visu;
END_STRUCT
END_TYPE

(* Data type in Gemeinsamkeiten17xx/Haspel *)
TYPE struct_haspelkontroller :
STRUCT
	t_abschaltzeit_motor			: TIME := t#0s;
	b_drehrichtung_antrieb_links	: BOOL := FALSE;
	st_config						: struct_config;
	haspel1_ctrl_in				: struct_ctrl_out;
	haspel2_ctrl_in				: struct_ctrl_out;
	st_ctrl						: struct_ctrl;
	st_visu						: struct_visu;
	haspel1_ctrl_out				: struct_ctrl_in;
	haspel2_ctrl_out				: struct_ctrl_in;
END_STRUCT
END_TYPE

(* Data type in Gemeinsamkeiten17xx/Nockenschaltwerk *)
TYPE enum_nocken_namen :
	( NO_OT := 0,
	NO_START_SKALIERUNG,
	NO_VERFAHRFREIGABE_Z_ACHSE,
	NO_BW_BANDFAENGER_EINFAHREN,
	NO_BW_BANDFAENGER_AUSFAHREN,
	NO_BW_BANDKLEMMEN_EINFAHREN,
	NO_BW_BANDKLEMMEN_AUSFAHREN,
	NO_UW_BANDFAENGER_EINFAHREN,
	NO_UW_BANDFAENGER_AUSFAHREN,
	NO_UW_BANDKLEMMEN_EINFAHREN,	(* 9 *)
	NO_UW_BANDKLEMMEN_AUSFAHREN,
	NO_PRUEFE_BANDENDE_AM_EINZUG,
	NO_BESTUECKSCHIEBERHUB,
	NO_UW_BESTUECKSCHIEBER_ON,
	NO_UW_BESTUECKSCHIEBER_OFF,
	NO_AUFNAHMEHUB,
	NO_EINPRESSHUB,
	NO_BW_BANDFAENGER_LI_EINFAHREN,
	NO_BW_BANDFAENGER_LI_AUSFAHREN,
	NO_BW_BANDKLEMMEN_LI_EINFAHREN,	(* 19 *)
	NO_BW_BANDKLEMMEN_LI_AUSFAHREN,
	NO_UW_BANDFAENGER_LI_EINFAHREN,
	NO_UW_BANDFAENGER_LI_AUSFAHREN,
	NO_UW_BANDKLEMMEN_LI_EINFAHREN,
	NO_UW_BANDKLEMMEN_LI_AUSFAHREN,
	NO_BW_BANDFAENGER_RE_EINFAHREN,
	NO_BW_BANDFAENGER_RE_AUSFAHREN,
	NO_BW_BANDKLEMMEN_RE_EINFAHREN,
	NO_BW_BANDKLEMMEN_RE_AUSFAHREN,
	NO_UW_BANDFAENGER_RE_EINFAHREN,	(* 29 *)
	NO_UW_BANDFAENGER_RE_AUSFAHREN,
	NO_UW_BANDKLEMMEN_RE_EINFAHREN,
	NO_UW_BANDKLEMMEN_RE_AUSFAHREN,
	NO_UW_WKZ_NIEDERHALTER_LI,
	NO_UW_WKZ_NIEDERHALTER_RE,
	NO_PNEUMATIKBANDEINZUG_GLS,
	NO_BW_BANDFAENGER_BAWEV2_EINFAHREN,
	NO_BW_BANDFAENGER_BAWEV2_AUSFAHREN,
	NO_BW_BANDKLEMMEN_BAWEV2_EINFAHREN,
	NO_BW_BANDKLEMMEN_BAWEV2_AUSFAHREN,	(* 39 *)
	NO_BW_BANDFAENGER_LI_BAEZV2_EINFAHREN,
	NO_BW_BANDFAENGER_LI_BAEZV2_AUSFAHREN,
	NO_BW_BANDKLEMMEN_LI_BAEZV2_EINFAHREN,
	NO_BW_BANDKLEMMEN_LI_BAEZV2_AUSFAHREN,
	NO_BW_BANDFAENGER_RE_BAEZV2_EINFAHREN,
	NO_BW_BANDFAENGER_RE_BAEZV2_AUSFAHREN,
	NO_BW_BANDKLEMMEN_RE_BAEZV2_EINFAHREN,
	NO_BW_BANDKLEMMEN_RE_BAEZV2_AUSFAHREN,
	NO_SERVOBANDEINZUG_LUEFTEN,
	NO_SERVOBANDEINZUG_GLS,
	NO_MIN_KRAFT_EINPRESSEN := 50,
	NO_BW_BESTUECKSCHIEBER_EINSTEUERN,
	NO_UW_BESTUECKSCHIEBER_EINSTEUERN,
	NO_DISABLE_AUTO_RESET,
	NO_RASTERFOLIE_LUEFTEN);
END_TYPE

(* Data type in Gemeinsamkeiten17xx/Nockenschaltwerk *)
TYPE enum_spur_namen :
	( SP_OT := 0,
	SP_START_SKALIERUNG,
	SP_VERFAHRFREIGABE_Z_ACHSE,
	SP_BW_BANDFAENGER_EINFAHREN,
	SP_BW_BANDFAENGER_AUSFAHREN,
	SP_BW_BANDKLEMMEN_EINFAHREN,
	SP_BW_BANDKLEMMEN_AUSFAHREN,
	SP_UW_BANDFAENGER_EINFAHREN,
	SP_UW_BANDFAENGER_AUSFAHREN,
	SP_UW_BANDKLEMMEN_EINFAHREN,
	SP_UW_BANDKLEMMEN_AUSFAHREN,
	SP_PRUEFE_BANDENDE_AM_EINZUG,
	SP_BESTUECKSCHIEBERHUB,
	SP_UW_BESTUECKSCHIEBER_ON,
	SP_UW_BESTUECKSCHIEBER_OFF,
	SP_AUFNAHMEHUB,
	SP_EINPRESSHUB,
	SP_BW_BANDFAENGER_LI_EINFAHREN,
	SP_BW_BANDFAENGER_LI_AUSFAHREN,
	SP_BW_BANDKLEMMEN_LI_EINFAHREN,
	SP_BW_BANDKLEMMEN_LI_AUSFAHREN,
	SP_UW_BANDFAENGER_LI_EINFAHREN,
	SP_UW_BANDFAENGER_LI_AUSFAHREN,
	SP_UW_BANDKLEMMEN_LI_EINFAHREN,
	SP_UW_BANDKLEMMEN_LI_AUSFAHREN,
	SP_BW_BANDFAENGER_RE_EINFAHREN,
	SP_BW_BANDFAENGER_RE_AUSFAHREN,
	SP_BW_BANDKLEMMEN_RE_EINFAHREN,
	SP_BW_BANDKLEMMEN_RE_AUSFAHREN,
	SP_UW_BANDFAENGER_RE_EINFAHREN,
	SP_UW_BANDFAENGER_RE_AUSFAHREN,
	SP_UW_BANDKLEMMEN_RE_EINFAHREN,
	SP_UW_BANDKLEMMEN_RE_AUSFAHREN,
	SP_UW_WKZ_NIEDERHALTER_LI,
	SP_UW_WKZ_NIEDERHALTER_RE,
	SP_PNEUMATIKBANDEINZUG_GLS,
	SP_BW_BANDFAENGER_BAWEV2_EINFAHREN,
	SP_BW_BANDFAENGER_BAWEV2_AUSFAHREN,
	SP_BW_BANDKLEMMEN_BAWEV2_EINFAHREN,
	SP_BW_BANDKLEMMEN_BAWEV2_AUSFAHREN,
	SP_BW_BANDFAENGER_LI_BAEZV2_EINFAHREN,
	SP_BW_BANDFAENGER_LI_BAEZV2_AUSFAHREN,
	SP_BW_BANDKLEMMEN_LI_BAEZV2_EINFAHREN,
	SP_BW_BANDKLEMMEN_LI_BAEZV2_AUSFAHREN,
	SP_BW_BANDFAENGER_RE_BAEZV2_EINFAHREN,
	SP_BW_BANDFAENGER_RE_BAEZV2_AUSFAHREN,
	SP_BW_BANDKLEMMEN_RE_BAEZV2_EINFAHREN,
	SP_BW_BANDKLEMMEN_RE_BAEZV2_AUSFAHREN,
	SP_SERVOBANDEINZUG_LUEFTEN,
	SP_SERVOBANDEINZUG_GLS,
	SP_MIN_KRAFT_EINPRESSEN := 50,
	SP_BW_BESTUECKSCHIEBER_EINSTEUERN,
	SP_UW_BESTUECKSCHIEBER_EINSTEUERN,
	SP_DISABLE_AUTO_RESET,
	SP_RASTERFOLIE_LUEFTEN);
END_TYPE

(* Data type in Gemeinsamkeiten17xx/Oeler *)
TYPE struct_bandoeler :
STRUCT
	fb			: ST_Bandoeler;
	st_ctrl		: struct_ctrl;
END_STRUCT
END_TYPE

(* Data type in Gemeinsamkeiten17xx/Oeler *)
TYPE struct_oeler :
STRUCT
	i16_intervall_bandoelen				: INT := 1;
	t_ventiloeffnungszeit					: DINT := 500;
END_STRUCT
END_TYPE

(* Data type in Gemeinsamkeiten17xx/Oeler *)
TYPE struct_oeler_daten :
STRUCT
	i32_neue_intervallvorgabe		: DINT := 500;
	t_ventiloeffnungszeit			: TIME := t#10ms;
	t_oelzeit_nach_stillstand		: TIME := t#20ms;
	i32_aktueller_stand			: DINT := 0;
	i32_alte_intervallvorgabe		: DINT := 0;
END_STRUCT
END_TYPE

(* Data type in Gemeinsamkeiten17xx/Oeler *)
TYPE struct_oeler_retain :
STRUCT
	i32_neue_intervallvorgabe		: DINT := 500;
	t_ventiloeffnungszeit			: TIME := t#10ms;
	t_oelzeit_nach_stillstand		: TIME := t#20ms;
	i32_aktueller_stand			: DINT := 0;
	i32_alte_intervallvorgabe		: DINT := 0;
END_STRUCT
END_TYPE

(* Data type in Gemeinsamkeiten17xx/Oeler *)
TYPE struct_oeler_visu :
STRUCT
	b_handoelen							: BOOL := FALSE;
END_STRUCT
END_TYPE

(* Data type in Gemeinsamkeiten17xx/Oeler *)
TYPE struct_schmier_daten :
STRUCT
	i32_neue_intervallvorgabe		: DINT := 500;
	t_ventiloeffnungszeit			: TIME := t#10ms;
	i32_aktueller_stand			: DINT := 0;
	i32_alte_intervallvorgabe		: DINT := 0;
END_STRUCT
END_TYPE

(* Data type in Gemeinsamkeiten17xx/Stueckzahlen *)
TYPE enum_zaehlerart :
	(
	JAHR := 0,
	AUFTRAG,
	VPE
	);
END_TYPE

(* Data type in Gemeinsamkeiten17xx/Stueckzahlen *)
TYPE struct_gut_schlecht_teile :
STRUCT
	i32_aktuelle_gutteile		: DINT := 0;
	i32_aktuelle_schlechtteile	: DINT := 0;
	i32_vorgabe_gutteile		: DINT := 0;
	b_reset_gutteile			: BOOL := FALSE;
	b_reset_schlechtteile		: BOOL := FALSE;
END_STRUCT
END_TYPE

(* Data type in Gemeinsamkeiten17xx/Stueckzahlen *)
TYPE struct_stueckzahl :
STRUCT
	fb			: ST_Stueckzahl;
	st_ctrl		: struct_ctrl;
END_STRUCT
END_TYPE

(* Data type in Gemeinsamkeiten17xx/Stueckzahlen *)
TYPE struct_stueckzahlen :
STRUCT
	st_teilezaehler		: ARRAY[0..2] OF struct_gut_schlecht_teile;
END_STRUCT
END_TYPE

(* Data type in Gemeinsamkeiten17xx/Tag_Reader *)
TYPE enum_part_state :
(
(*	PART_UNDEFINDED		:= -1, (*State not defined*)*)
	PART_NO				:= 0, (*no Part available*)
	PART_OK				:= 1, (*Part processed with OK-Result*)
	PART_NOK				:= 2, (*Part processed with NOK-Result*)
	PART_NEW			:= 4,  (*new Part (picked up from Feeder, and not yet processed) *)
	PART_DUMMY			:= 99, (*dummy Part on Wpc *)
	XXXX					:= 100 (*Tag lesen*)
);
END_TYPE

(* Data type in Gemeinsamkeiten17xx/Tag_Reader *)
TYPE struct_tag_data :
STRUCT
	WpcNumber			: BYTE;
	StateParts				: ARRAY[0..7] OF enum_part_state;
	AmountPartsOnWpc		: BYTE;
	LastUsedTool			: BYTE;
	Articelnumber			: STRING(50);
	UmlNo_VPE				: DINT:=100;  	(*erste Zahl immer 1 + UMl-Nummer max 99   danach max 6 Stellen für VPE =>  z.B. 1 78 100123  wird für die automatisch LTS buchung benutzt*)
END_STRUCT
END_TYPE

(* Data type in Gemeinsamkeiten17xx/Visu *)
TYPE struct_servobandeinzug :
STRUCT
	b_taste_bremse				: BOOL := FALSE;
	b_taste_tippen				: BOOL := FALSE;
END_STRUCT
END_TYPE

(* Data type in Gemeinsamkeiten17xx/Visu *)
TYPE struct_taste_ein_aus :
STRUCT
	b_einfahren				: BOOL := FALSE;
	b_ausfahren				: BOOL := FALSE;
END_STRUCT
END_TYPE

(* Data type in Gemeinsamkeiten17xx/Visu *)
TYPE struct_texte :
STRUCT
	txt_zylindernamen	: ARRAY [0..16] OF struct_zyltexte_ein_aus;
	txt_statisch			: ARRAY [0..35] OF STRING(255) := '';
	txt_variabel			: ARRAY [0..15] OF STRING(255) := '';
	txt_bm_einfaedeln	: ARRAY [0..15] OF STRING(255) := '';
END_STRUCT
END_TYPE

(* Data type in Gemeinsamkeiten17xx/Visu *)
TYPE struct_visu :
STRUCT
	b_quittieren								: BOOL := FALSE;
	b_start									: BOOL := FALSE;
	b_stop									: BOOL := FALSE;
	b_einzelfertigung							: BOOL := FALSE;
	b_tippen_start							: BOOL := FALSE;
	b_start_foerderband						: BOOL := FALSE;
	b_inbetriebnahme							: BOOL := FALSE;
	b_geschwindigkeit_vorgabe				: BOOL := FALSE;
	b_vollbestuecken							: BOOL := FALSE;
	b_merker_vollbestuecken					: BOOL := FALSE;
	b_Reset_Band_ID							: BOOL := FALSE;
	b_handoelen								: BOOL := FALSE;
	b_reset_wartung_wkz						: BOOL := FALSE;
	b_reset_wartung_maschine					: BOOL := FALSE;
	s_akt_sprache							: STRING(255) := 'de';
	st_nocken								: struct_nocken_visu;
	st_zyl									: struct_zylinder_visu;
	st_achsen								: ARRAY [0..3] OF struct_ecd_visu;
	st_xml_server								: struct_xml_visu;
	st_tagreader								: struct_visu_tagreader;
	st_service								: struct_visu_service;
	st_bandwechsler							: struct_bandwechsler_visu;
	MeldungProduktion	 					: struct_MeldungProduktion;
	b_logon									: BOOL;
	b_start_remove_pos						: BOOL;
	b_save									: BOOL := FALSE;
	b_load									: BOOL := FALSE;
	b_fbwf_info								: BOOL := FALSE;
	b_fbwf_disable							: BOOL := FALSE;
	b_fbwf_enable							: BOOL := FALSE;
END_STRUCT
END_TYPE

(* Data type in Gemeinsamkeiten17xx/Visu *)
TYPE struct_visu_hinten :
STRUCT
	in	:	struct_visu_hinten_in;
	out	:	struct_visu_hinten_out;
END_STRUCT
END_TYPE

(* Data type in Gemeinsamkeiten17xx/Visu *)
TYPE struct_visu_hinten_in :
STRUCT
	betriebsart				: STRING(255) := '';
	s_maschinenstatusinfo 		: STRING(255) := '';
	i16_maschinenstatusinfo	: INT := 0;
	s_betriebsmeldung		: STRING(255) := '';
	i16_position_ist			: INT := 0;
	zylinder_sensoren			: ARRAY [0..16] OF struct_zylinder_sensoren;
	texte					: struct_texte;
	bandfreigabe				: ARRAY [0..1] OF BOOL;
	band_ID					: ARRAY [0..1] OF BOOL;
	scannen_moeglich		: ARRAY [0..1] OF BOOL;
	i16_typ_zelle				: enum_typ_zelle := KEINE_ZELLE;
	i16_typ_bandeinzug		: enum_typ_bandeinzug := KEIN_EINZUG;
	s_aktuelles_wkz			: STRING(50);
	s_Barcode				: STRING(50);
	s_aktuelles_band			: STRING(50);
	b_zustand_bremse		: BOOL := FALSE;
	current_visu_folie			: STRING(50);
	b_bandwechsel_aktiv		: BOOL := FALSE;
	sm_Meldung				: ARRAY [0..14] OF STRING(255);
	bm_Meldung				: ARRAY [0..14] OF STRING(255);
	band_ID_Puffer_aus		: BOOL := FALSE;
	Lampe_auto_Bandwechsel	: BOOL := FALSE;
END_STRUCT
END_TYPE

(* Data type in Gemeinsamkeiten17xx/Visu *)
TYPE struct_visu_hinten_out :
STRUCT
	zylinder_direkttasten			: ARRAY [0..16] OF struct_taste_ein_aus;		(* Direkttasten für Haspelzylinder u.s.w. *)
	b_quittieren					: BOOL := FALSE;
	b_start						: BOOL := FALSE;
	b_stop						: BOOL := FALSE;
	b_einzelfertigung				: BOOL := FALSE;
	b_tippen						: BOOL := FALSE;
	b_Bandwechsel				: BOOL;
	b_Trennstelle					: BOOL;
	auto_Bandwechsel_aus		: BOOL;
	st_servobandeinzug			: struct_servobandeinzug;
END_STRUCT
END_TYPE

(* Data type in Gemeinsamkeiten17xx/Visu *)
TYPE struct_visu_service :
STRUCT
	t_WT_wechsel					:TIME;
	t_Zentrierer_ausfahren			:TIME;
	t_Z_Achse_einfahren			:TIME;
	t_Bestueckung					:TIME;
	t_Z_Achse_ausfahren			:TIME;
	t_Zentrierer_einfahren			:TIME;

	t_Traegerwechselzeit			:TIME;
	t_komplett_zyklus				:TIME;
END_STRUCT
END_TYPE

(* Data type in Gemeinsamkeiten17xx/Visu *)
TYPE struct_visu_tagreader :
STRUCT
	b_start_lesen								: BOOL := FALSE;
	b_start_schreiben							: BOOL := FALSE;
	b_tag_im_Aktionsfeld						: BOOL;
	b_WT_ruecksetzen						: BOOL := FALSE;

	Farbwechsel								:ARRAY [1..12] OF BOOL;
END_STRUCT
END_TYPE

(* Data type in Gemeinsamkeiten17xx/Visu *)
TYPE struct_zylinder_sensoren :
STRUCT
	b_eingefahren		: BOOL := FALSE;
	b_ausgefahren		: BOOL := FALSE;
END_STRUCT
END_TYPE

(* Data type in Gemeinsamkeiten17xx/Visu *)
TYPE struct_zyltexte_ein_aus :
STRUCT
	s_einfahren	: STRING(255) := '';
	s_ausfahren	: STRING(255) := '';
END_STRUCT
END_TYPE

(* Data type in Gemeinsamkeiten17xx/Wartung *)
TYPE struct_Wartungsprotokoll :
STRUCT
	st_wartung_md	: struct_Wartungsprotokoll_md;
	st_wartung_wkz	: struct_Wartungsprotokoll_wkz;
END_STRUCT
END_TYPE

(* Data type in Gemeinsamkeiten17xx/Wartung *)
TYPE struct_Wartungsprotokoll_md :
STRUCT
	hubzaehler			: UDINT;
	produzierte_stecker	: UDINT;
	betriebsstunden		: LREAL;
END_STRUCT
END_TYPE

(* Data type in Gemeinsamkeiten17xx/Wartung *)
TYPE struct_Wartungsprotokoll_wkz :
STRUCT
	hubzaehler			: UDINT;
END_STRUCT
END_TYPE

(* Data type in Gemeinsamkeiten17xx/XML_Server *)
TYPE enum_xml_auftrag :
	(
	KEIN := 0,
	WKZ_WECHSELN,
	WKZ_SPEICHERN,
	WKZ_LADEN,
	WKZ_KOPIEREN,
	WKZ_EINLESEN,
	MD_SPEICHERN,
	MD_LADEN
	);
END_TYPE

(* Data type in Gemeinsamkeiten17xx/XML_Server *)
TYPE struct_xml_visu :
STRUCT
	b_taste_daten_speichern			: BOOL := FALSE;
	b_taste_daten_laden				: BOOL := FALSE;
	b_taste_daten_kopieren			: BOOL := FALSE;
	b_taste_daten_einlesen			: BOOL := FALSE;
	i16_quelldatensatz					: INT := 0;
	i16_zieldatensatz					: INT := 0;
END_STRUCT
END_TYPE

(* Data type in Maschine1700/Band *)
TYPE struct_bandwechsler :
STRUCT
	st_config		: struct_config;
	st_ctrl		: struct_ctrl;
	st_visu		: struct_visu;
END_STRUCT
END_TYPE

(* Data type in Maschine1700/Band *)
TYPE struct_bandwechsler_visu :
STRUCT
	b_taste_io			: BOOL := FALSE;
	b_taste_nio			: BOOL := FALSE;
END_STRUCT
END_TYPE

(* Data type in Maschine1700/Einpresskraftueberwachung *)
TYPE enum_einpressmodus :
	(
	KEIN_MODUS := 0,
	F_MAXWERT,
	F_MITTELWERT
	);
END_TYPE

(* Data type in Maschine1700/Einpresskraftueberwachung *)
TYPE struct_einpressausgabe :
STRUCT
	st_ergebnisse					: struct_weg_kraft_ergebnisse;
	st_kurve							: ARRAY[0..99] OF struct_kurven;
END_STRUCT
END_TYPE

(* Data type in Maschine1700/Einpresskraftueberwachung *)
TYPE struct_einpresskraftueberwachung :
STRUCT
	st_einstellungen			: struct_weg_kraft_einstellungen;
END_STRUCT
END_TYPE

(* Data type in Maschine1700/Einpresskraftueberwachung *)
TYPE struct_kurven :
STRUCT
	arr_weg_stuetz			: ARRAY[0..360] OF LREAL;
	arr_kraft_stuetz			: ARRAY[0..360] OF LREAL;
	arr_weg_ist				: ARRAY[0..360] OF LREAL;
	arr_kraft_ist				: ARRAY[0..360] OF LREAL;
END_STRUCT
END_TYPE

(* Data type in Maschine1700/Einpresskraftueberwachung *)
TYPE struct_weg_kraft_einstellungen :
STRUCT
	enu_modus				: enum_einpressmodus := F_MAXWERT;
	lr_maxkraft_aufnahme		: LREAL := 0;
	lr_maxkraft_einpressen		: LREAL := 100;
	lr_minkraft_einpressen		: LREAL := 0;
	lr_delta_kraft				: LREAL := 20;
	lr_delta_weg				: LREAL := 0;
END_STRUCT
END_TYPE

(* Data type in Maschine1700/Einpresskraftueberwachung *)
TYPE struct_weg_kraft_ergebnisse :
STRUCT
	lr_reserve				: LREAL := 0;
	lr_maxkraft_einpressen		: LREAL := 0;
	lr_maxkraft_einpres_proHub: LREAL := 0;
	lr_ueberlaufkraft			: LREAL := 0;
	lr_minkraft_einpressen		: LREAL := 0;
	lr_maxkraft_aufnahme		: LREAL := 0;
END_STRUCT
END_TYPE

(* Data type in Rasterfolie/Rafo_BBGen *)
TYPE struct_daten_rasterfolie :
STRUCT
	lr_pruefpos_rafo					: LREAL := 0.0;	(*Abstand zwischen Bestückposition und Prüfposition*)
	lr_pos_absenken				: LREAL := 0.0;
END_STRUCT
END_TYPE

(* Data type in Rasterplatte/Rapl_BBGen *)
TYPE struct_daten_rasterplatte :
STRUCT
	lr_anfang_pruefpos_rapl		: LREAL := 20.0;
	lr_ende_pruefpos_rapl			: LREAL := 30.0;
	lr_pos_absenken				: LREAL := 0.0;
	lr_pruefpos_rastnase_z			: ARRAY  [0..2] OF LREAL := 0.0;
	lr_pruefpos_rastnase_y		: ARRAY  [0..2] OF LREAL := 0.0;
END_STRUCT
END_TYPE

(* Data type in Visu/ButtonVisu *)
TYPE struct_ButtonVisu :
STRUCT
		sichtbar						: BOOL;
		tasten						: BOOL;
		Text							: STRING(30);
END_STRUCT
END_TYPE

(* Data type in Visu/EtherCatDiagnose *)
TYPE struct_EthercatDiagnose :
STRUCT
	st_Master			: struct_EthercatMaster;
	st_Slave			: ARRAY[1..MaxNoOfSlaves] OF struct_EthercatSlave;

END_STRUCT
END_TYPE

(* Data type in Visu/EtherCatDiagnose *)
TYPE struct_EthercatMaster :
STRUCT
	s_Name				: STRING := 'Master undefined';	(*Name des Ethercat Masters*)
	s_AmsNetId			: STRING := '0.0.0.0.0.0';			(*AmsNetId des Ethercat Masters*)
	i_Slaves				: INT := 0;							(*Anzahl konfigurierter Slaves*)
	f_FramesPerSeconed	: LREAL := 0;
	i_LostFrames			: UDINT := 0;
END_STRUCT
END_TYPE

(* Data type in Visu/EtherCatDiagnose *)
TYPE struct_EthercatSlave :
STRUCT
	i_Number			: INT;		(*Nummer in Ethercat Strang*)
	s_DeviceState		: STRING;	(*z.B. INIT, OP*)
	s_Name			: STRING;	(*Konfigurierter Name z.B. CO1_EL6910*)
	s_Type				: STRING;	(*z.B. EL6910*)
	s_Adress			: STRING;	(*Ethercat Adresse z.B. 1003*)
	b_Err				: BOOL;		(*nicht OP*)
END_STRUCT
END_TYPE

(* Data type in Visu *)
TYPE sMessageLine :
STRUCT
	MsgString		: STRING(40);
END_STRUCT
END_TYPE

(* Data type in Visu *)
TYPE struct_MeldungProduktion :
STRUCT
	ShowMessage				: BOOL;
	Name						: STRING(250);
	Text						: ARRAY [0..9] OF STRING(250);
	Color_R						: INT;
	Color_G						: INT;
	Color_B						: INT;

	Button1						: struct_ButtonVisu;
	Button2						: struct_ButtonVisu;

END_STRUCT
END_TYPE

(* Data type *)
TYPE enum_typ_achse :
	(
	BECKHOFF := 0,
	FESTO
	);
END_TYPE

(* Data type *)
TYPE enum_wartung_auftrag :
(
	KEIN_WARTUNG_AUFTRAG := 0,
	LESE_WARTUNGSPROTOKOLL_WKZ,
	LESE_WARTUNGSPROTOKOLL_MD,
	LESE_WARTUNGSPROTOKOLL_KOMPLETT,
	SCHREIBE_WARTUNGSPROTOKOLL_WKZ,
	SCHREIBE_WARTUNGSPROTOKOLL_WKZ_RESET,
	SCHREIBE_WARTUNGSPROTOKOLL_MD,
	SCHREIBE_WARTUNGSPROTOKOLL_KOMPLETT,
	SPEICHERN_WARTUNGSPROTOKOLL
);
END_TYPE

(* POU EPT Lib/Daten/ST_AutoCheckIn, ST *)
PROGRAM ST_AutoCheckIn
VAR_INPUT
	st_ctrl_in				: struct_ctrl_in;
	fb_AutocheckinDaten	: FB_StartWinProcess;
	i_IntervalDay				: INT;		(*all  X Tagen, 0 = jeden Tag*)
END_VAR
VAR_OUTPUT
	st_ctrl_out				: struct_ctrl_out;
END_VAR
VAR
	fb_state_entry			:ST_StateEntry;
	fb_ton_quitt				:TON;

	str_uhrzeit				:STRING;
	i_DayOfYear			:DINT;
	s_infoFile				:STRING;
	s_ScriptFile				:STRING;

END_VAR

VAR CONSTANT
		s_AutoCheckInMDtxt				:STRING:=		'AutoCheckInMD.txt';
		s_AutoCheckInMDBat				:STRING:=		'AutoCheckInMD.bat';

END_VAR
(*======================================================
   FB: Start eines Win Prozess mit Prüfung 
 ------------------------------------------------------
   Auth: 		Werner Friedl   						 
   Date: 		19.02.2019   						     
   Rev.: 		1.0	
   Desc:		Mit diesem Programm Können Komponenten im Versdog automatisch eingecheckt werden.
			Für den Check in benötigt man einen Bat- Datei. Diese liegt im Projektverzeichniss "Tools" und 
			muss für jede Komponente erstellt werden.
			Wenn mehrere Komponeten Eingecheckt werden sollen muss der Schritt 110 bis 120 mehrfach
			ausgefühtr werden.

			- die Input Variable "i16_Intervall" legt den Seicherintervall in x Tagen fest.
			Wenn das Speichern nicht klappt, dann wird einen Tag später der nächste Versuch gemacht.

   Historie:   1.0

=======================================================*)

(* Zeiten *)
fb_ton_quitt(IN:= , PT:= t#100ms, Q=> , ET=> );

(* Tag im Jahr *)
i_DayOfYear:=F_GetDOYOfYearMonthDay( gst_system_time.wYear, gst_system_time.wMonth, gst_system_time.wDay );

fb_state_entry(i16_pos:= 1);

CASE fb_state_entry.i16_step OF

(*=======================================================*)
INIT_OBJ:

	(*-----------------------Weiterschaltbedingungen----------------------------*)
	IF	gst_datensatz.st_md.i16_typ_zelle <> KEINE_ZELLE AND
		gstr_uhrzeit <> '00:00:00' AND gstr_uhrzeit <> ''  THEN
		IF	gst_PersDaten.i_DayOfYearAutoCheckIn > i_DayOfYear THEN
			gst_PersDaten.i_DayOfYearAutoCheckIn:= i_DayOfYear;
		END_IF
			fb_state_entry.i16_next_step := 5;
	END_IF

(*=======================================================*)
5:
	IF fb_state_entry.E THEN
		str_uhrzeit:=gstr_uhrzeit;
		(*str_uhrzeit:=REPLACE (str_uhrzeit,'00',2,1);*)	(*nur in der Nacht sichern*)
	END_IF

	(*-----------------------Weiterschaltbedingungen----------------------------*)
	IF 	fb_state_entry.fb_ton_Step.ET > t#59s THEN
		IF	gst_PersDaten.i_DayOfYearAutoCheckIn + i_IntervalDay < i_DayOfYear  THEN
			fb_state_entry.i16_next_step:=110;		(*gleich sicher, da das letzte Sichern zu lange her ist*)
		ELSE
			fb_state_entry.i16_next_step:=INIT;
		END_IF
	END_IF

(*=======================================================*)
INIT:
	IF fb_state_entry.E THEN
		fb_ton_quitt.IN := FALSE;
		st_ctrl_out.b_fehler := FALSE;
		st_ctrl_out.b_gestoppt := FALSE;
		st_ctrl_out.b_bereit := FALSE;
		st_ctrl_out.b_fertig := FALSE;
		st_ctrl_out.b_busy := FALSE;
	END_IF

	(*-----------------------Weiterschaltbedingungen----------------------------*)
	fb_state_entry.i16_next_step := BEREIT;

(*=======================================================*)
BEREIT: fb_state_entry.s_debugtext:='warte auf Start';

	IF fb_state_entry.E THEN
		st_ctrl_out.b_bereit:=TRUE;
	END_IF

	(*-----------------------Weiterschaltbedingungen----------------------------*)
	IF 	str_uhrzeit=gstr_uhrzeit AND
		(gst_PersDaten.i_DayOfYearAutoCheckIn + i_IntervalDay) <= i_DayOfYear THEN
		fb_state_entry.i16_next_step:=110;
	END_IF

	IF fb_state_entry.X THEN
		st_ctrl_out.b_busy:=TRUE;
		st_ctrl_out.b_bereit := FALSE;
		st_ctrl_out.b_fertig := FALSE;
	END_IF

(*=======================================================*)
110:  fb_state_entry.s_debugtext:='Start Autocheckin';

	IF fb_state_entry.E THEN
		s_infoFile:=s_AutoCheckInMDtxt;
		s_ScriptFile:=s_AutoCheckInMDBat;
		fb_AutocheckinDaten.st_ctrl_in.b_start:=TRUE;
	END_IF

	(*-----------------------Weiterschaltbedingungen----------------------------*)
	IF	fb_AutocheckinDaten.st_ctrl_out.b_busy THEN
		fb_state_entry.i16_next_step:=120;
	ELSIF	fb_state_entry.fb_ton_Step.ET > t#15s THEN
		fb_state_entry.i16_next_step:=FEHLER;
	END_IF

(*=======================================================*)
120:  fb_state_entry.s_debugtext:='Warte auf fertig Autocheckin';

	(*-----------------------Weiterschaltbedingungen----------------------------*)
	IF	fb_AutocheckinDaten.st_ctrl_out.b_fertig THEN
		fb_state_entry.i16_next_step:=200;
	ELSIF
		fb_state_entry.fb_ton_Step.ET > t#59s OR
		fb_AutocheckinDaten.st_ctrl_out.b_fehler THEN
		fb_state_entry.i16_next_step:=FEHLER;
		gst_PersDaten.i_DayOfYearAutoCheckIn:=i_DayOfYear - i_IntervalDay+1; (*bei einem Fehler wird die nächst Sicherung einen Tag später nochmal gemacht*)
	END_IF

(*=======================================================*)
200:  fb_state_entry.s_debugtext:='Ende';

	(*-----------------------Weiterschaltbedingungen----------------------------*)
	fb_state_entry.i16_next_step:=BEREIT;
	gst_PersDaten.i_DayOfYearAutoCheckIn:=i_DayOfYear;
	IF fb_state_entry.X THEN
		st_ctrl_out.b_busy:=FALSE;
		st_ctrl_out.b_fertig := TRUE;
	END_IF

(*=======================================================*)
STOP, FEHLER:
	IF fb_state_entry.E THEN
		st_ctrl_out.b_fehler := fb_state_entry.i16_step = FEHLER;
		st_ctrl_out.b_gestoppt := fb_state_entry.i16_step = STOP;
		fb_ton_quitt.IN := FALSE;
		st_ctrl_out.b_busy:=FALSE;
		st_ctrl_out.b_fertig:=FALSE;
		fb_ton_quitt.IN := TRUE;				(*quttiert sich selbst*)
	END_IF

	(*-----------------------Weiterschaltbedingungen----------------------------*)
	IF 	st_ctrl_in.b_quitt THEN
		fb_ton_quitt.IN := TRUE;
	END_IF

	IF fb_ton_quitt.Q THEN
		fb_ton_quitt.IN := FALSE;
		st_ctrl_out.b_fehler := FALSE;
		fb_state_entry.i16_next_step := INIT;
	END_IF

END_CASE

fb_state_entry(i16_pos:= 2 );
st_ctrl_in:=st_ctrl_in_empty;


(*Aufrufe======================================================*)
fb_AutocheckinDaten(
	s_path:= 			s_tools_path,								(*Verzeichnis der bat,vbs und Prüf- Datei*)
	s_info_file:=			CONCAT(s_tools_path,s_infoFile) ,			(*Datei in der die Prüfung landet*)
	s_script:=			s_ScriptFile ,								(*auszuführende Datei bat oder vbs eintragen*)
	i16_Timeout:= 	100);											(*in sec*)
END_PROGRAM

(* POU EPT Lib/Daten/FB_StartWinProcess, ST *)
FUNCTION_BLOCK FB_StartWinProcess
VAR_INPUT
	st_ctrl_in			:struct_ctrl_in;
	st_config			: struct_config;
	s_path				:STRING(255);		(*Pfad der Bat- oder vbs- Datei*)
	s_info_file			:STRING(255);		(*Pfad + Dateiname der Statusdatei*)
	s_script				:STRING;
	i16_Timeout			:INT;			(*in sec*)
	b_Start				:BOOL;
END_VAR
VAR_OUTPUT
	st_ctrl_out				:struct_ctrl_out;
	ErrId					:UDINT;
	ErrTyp					:STRING(5);
	ErrorMsg				:STRING(255);
	MsgString				:STRING(255);
END_VAR
VAR
	b_init					:BOOL;
	fb_state_entry			:ST_StateEntry;

	NT_StartProcess 		:NT_StartProcess;
	fbFileOpen				:FB_FileOpen;
	fbFileRead				:FB_FileRead;
	fbFileClose				:FB_FileClose;
	fbFileDelete				:FB_FileDelete;
	hFile					:UINT;

	fb_ton_wz				:TON;
	fb_ton_quitt				:TON;
	pos						:INT;
	FileString				:STRING(255);
	i16_Time				:INT;	(*in sec*)
	i						:INT;
	b_sm					:ARRAY[0..9] OF BOOL;	(*Störmeldungen aus der bat oder vbs Datei*)
	b_bm					:ARRAY[0..9] OF BOOL;	(*Bertiebsmeldungen aus der bat oder vbs Datei*)
	(*sonstige Meldungen*)
	sm_DateiNichtVorhanden				:BOOL;
	sm_FehlerBeimOeffnenDerDatei		:BOOL;
	sm_FehlerBeimAuslesenDerDatei		:BOOL;
	sm_FehlerBeimSchliessenDerDatei		:BOOL;
	sm_FehlerBeimLoeschenDerDatei		:BOOL;
	sm_KeineImportdateiVorhanden		:BOOL;
	sm_KeineErrIdGefunden				:BOOL;
END_VAR
(*======================================================
   FB: Start eines Win Prozess mit Prüfung 
 ------------------------------------------------------
   Auth: 		Werner Friedl   						 
   Date: 		19.02.2019   						     
   Rev.: 		1.0	
   Desc:		Eine Bat- oder vbs- Datei kann gestartet weden und der Status kommt über die ErrId wieder zurück.
			Die "ErrId" wird dann b_sm[ErrId] oder b_bm[ErrId], Damit können Betriebs und Störmeldungen von der bat angezeigt werden. 
			alle Meldungen quittieren sich selbst
			b_bm[0] =	'OK',
			b_sm[1] =	Netzwerk nicht verbunden!
			b_sm[2] =	User nicht vorhanden oder Passwort falsch!
			b_sm[3] =	Verzeichnis nicht vorhanden!
			b_sm[4] =	Datei nicht vorhanden!

   Historie:   1.0

   Aufruf Beispiel:
	s_instanz_name:='test',
	s_path:= 		s_tools_path,			(*Verzeichnis der Bat- und Prüf- Datei*)
	s_info_file:=	CONCAT(s_tools_path,'Test.txt') ,	(*Datei in der die Prüfung landet (sollte so heißen wie die Bat-Datei)*)
	s_script:=		'Test.bat' ,				(*auszuführende Datei bat oder vbs eintragen*)
	i16_Timeout:= 100);					(*in sec*)

 ========================================================*)
IF	NOT b_init THEN
	b_Init:=TRUE;
END_IF
(* ========================================================*)
fb_ton_quitt(IN:= , PT:= t#100ms, Q=> , ET=> );

fb_state_entry(i16_pos:= 1);
CASE fb_state_entry.i16_step OF
(*=======================================================*)
INIT_OBJ:
		fb_state_entry.i16_next_step := INIT;

(*=======================================================*)
INIT:	(*initialisieren*)
	IF fb_state_entry.E THEN
		fb_ton_quitt.IN := FALSE;
		st_ctrl_out.b_fehler := FALSE;
		st_ctrl_out.b_gestoppt := FALSE;
		st_ctrl_out.b_bereit := FALSE;
		st_ctrl_out.b_fertig := FALSE;
		st_ctrl_out.b_busy := FALSE;

		sm_DateiNichtVorhanden:=FALSE;
		sm_FehlerBeimOeffnenDerDatei:=FALSE;
		sm_FehlerBeimAuslesenDerDatei:=FALSE;
		sm_FehlerBeimSchliessenDerDatei:=FALSE;
		sm_FehlerBeimLoeschenDerDatei:=FALSE;
		sm_KeineImportdateiVorhanden:=FALSE;
		sm_KeineErrIdGefunden:=FALSE;
		FOR i:=0 TO 9 DO
			b_sm[i]:=FALSE;
			b_bm[i]:=FALSE;
		END_FOR
	END_IF

	(*-----------------------Weiterschaltbedingungen----------------------------*)
	fb_state_entry.i16_next_step:=BEREIT;

(*=======================================================*)
BEREIT: fb_state_entry.s_debugtext:='warte auf start';

	IF fb_state_entry.E THEN
		st_ctrl_out.b_bereit:=TRUE;
	END_IF

	(*-----------------------Weiterschaltbedingungen----------------------------*)
	IF	st_ctrl_in.b_start THEN
		NT_StartProcess.START:=TRUE;
		fb_state_entry.i16_next_step:=110;
	END_IF

	IF fb_state_entry.X THEN
		i16_Time:=0;
		st_ctrl_out.b_busy:=TRUE;
		st_ctrl_out.b_bereit := FALSE;
		st_ctrl_out.b_fertig := FALSE;
		ErrId:=99;
		ErrorMsg:='';
		FileString:='';
		MsgString:='';
	END_IF

	IF 	fb_state_entry.X THEN
		NT_StartProcess.START:=FALSE;
	END_IF

(*=======================================================*)
110:  fb_state_entry.s_debugtext:='start Datei öffnen';

	IF	fb_state_entry.fb_ton_Step.ET > t#1s THEN
		fbFileOpen.sPathName:=s_info_file;
   		fbFileOpen.bExecute:=TRUE;
	END_IF

	(*-----------------------Weiterschaltbedingungen----------------------------*)
	IF 	fbFileOpen.bBusy THEN
		fb_state_entry.i16_next_step:=120;
	END_IF

	IF 	fb_state_entry.X THEN
		ErrorMsg:='';
		st_ctrl_out.b_fehler:=FALSE;
	END_IF

(*=======================================================*)
120:  fb_state_entry.s_debugtext:='warte auf fertig Datei öffnen';

	IF 	NOT fbFileOpen.bBusy AND fb_state_entry.i16_next_step=120 THEN
		fbFileOpen.bExecute:=FALSE;
		IF	NOT fbFileOpen.bError THEN
			fb_state_entry.i16_next_step:=130;
		ELSIF
			fb_state_entry.fb_ton_Step.ET > t#1000ms THEN

			IF	i16_Time<=i16_Timeout THEN (*Datei nicht vorhanden*)
				fb_state_entry.i16_next_step:=110;
				i16_Time:=i16_Time+1;
			ELSE
				ErrId:=fbFileOpen.nErrId;
				fb_state_entry.i16_next_step:=FEHLER;

				IF 	fbFileOpen.nErrId =1804 THEN (*Datei nicht vorhanden*)
					sm_DateiNichtVorhanden:=TRUE;
					ErrorMsg:='Info Datei nicht vorhanden';
				ELSE
					sm_FehlerBeimOeffnenDerDatei:=TRUE;
					ErrorMsg:='Fehler beim Öffnen der Datei.';
				END_IF

			END_IF

		END_IF
	END_IF

(*=======================================================*)
130:  fb_state_entry.s_debugtext:='Start String aus Datei auslesen';

	fbFileRead.bExecute:=TRUE;
	IF 	fbFileRead.bBusy THEN
		fb_state_entry.i16_next_step:=140;
	END_IF

(*=======================================================*)
140:  fb_state_entry.s_debugtext:='warte auf fertig String aus Datei auslesen';

	IF 	NOT fbFileRead.bBusy THEN
		fbFileRead.bExecute:=FALSE;
		IF 	fbFileRead.bError THEN
			ErrId:=fbFileRead.nErrId;
			fb_state_entry.i16_next_step:=FEHLER;
			sm_FehlerBeimAuslesenDerDatei:=TRUE;
			ErrorMsg:='Fehler beim Auslesen der Datei.';
		ELSE
			fb_state_entry.i16_next_step:=150;
		END_IF
	END_IF

(*=======================================================*)
150: fb_state_entry.s_debugtext:='start Datei schließen';

	fbFileClose.bExecute:=TRUE;
	IF 	fbFileClose.bBusy THEN
		fb_state_entry.i16_next_step:=160;
	END_IF

(*=======================================================*)
160: fb_state_entry.s_debugtext:='warte auf fertig Datei schließen';

	IF 	NOT fbFileClose.bBusy THEN
		fbFileClose.bExecute:=FALSE;
		IF 	fbFileClose.bError THEN
			ErrId:=fbFileClose.nErrId;
			fb_state_entry.i16_next_step:=FEHLER;
			sm_FehlerBeimSchliessenDerDatei:=TRUE;
			ErrorMsg:='Fehler beim Schließen der Datei.';
		ELSE
			fb_state_entry.i16_next_step:=190;
		END_IF
	END_IF

(*=======================================================*)
170: fb_state_entry.s_debugtext:='start Datei löschen';

	fbFileDelete.bExecute:=TRUE;
	fbFileDelete.sPathName:=s_info_file;
	IF 	fbFileDelete.bBusy THEN
		fb_state_entry.i16_next_step:=180;
	END_IF

(*=======================================================*)
180: fb_state_entry.s_debugtext:='warte auf fertig Datei löschen';

	IF 	NOT fbFileDelete.bBusy THEN
		fbFileDelete.bExecute:=FALSE;
		IF 	fbFileDelete.bError THEN
			ErrId:=fbFileDelete.nErrId;
			fb_state_entry.i16_next_step:=FEHLER;
			sm_FehlerBeimLoeschenDerDatei:=TRUE;
			ErrorMsg:='Fehler beim löschen der Datei.';
		ELSE
			fb_state_entry.i16_next_step:=190;
		END_IF
	END_IF

(*=======================================================*)
190: fb_state_entry.s_debugtext:='Auswertung';

	IF 	fb_state_entry.E THEN
		MsgString:=FileString;

		(*falls noch ein Text mitkommt*)
		pos:=0;
		pos:=FIND (MsgString,'$N');
		IF 	pos >0 THEN
			ErrTyp:=LEFT(MsgString,pos-1);
			ErrId:=STRING_TO_INT(DELETE(ErrTyp,2,1));
			MsgString:=DELETE(MsgString,LEN(MsgString)-pos+2,pos);
		END_IF

		pos:=0;
		pos:=FIND (MSGString,'$T');
		IF 	pos >0 THEN
			MsgString:=DELETE(MsgString,1,pos);
		END_IF

	END_IF

	IF	LEN(FileString) = 0 THEN
		fb_state_entry.i16_next_step:=FEHLER;
		sm_KeineImportdateiVorhanden:=TRUE;
		ErrorMsg:='Kein Importstring vorhanden.';
	ELSE
		IF	ErrId <>99 THEN
			IF	FIND(ErrTyp,'BM') > 0 THEN
				b_bm[ErrId]:=TRUE;
			ELSIF	FIND(ErrTyp,'SM') > 0 THEN
				b_sm[ErrId]:=TRUE;
			END_IF
			fb_state_entry.i16_next_step:=200;
		ELSE
			sm_KeineErrIdGefunden:=TRUE;
			ErrorMsg:='**Error Id not found**';
			fb_state_entry.i16_next_step:=FEHLER;
		END_IF
	END_IF

(*=======================================================*)
200: fb_state_entry.s_debugtext:='Fertig';

	IF	fb_state_entry.fb_ton_Step.ET >t#5s THEN
		IF	FIND(ErrTyp,'BM') > 0 THEN
			fb_state_entry.i16_next_step:=INIT;
			st_ctrl_out.b_fertig:=TRUE;
		ELSE
			fb_state_entry.i16_next_step:=FEHLER;
		END_IF

	END_IF

	IF fb_state_entry.X THEN
		st_ctrl_out.b_busy:=FALSE;
	END_IF

(*=======================================================*)
STOP, FEHLER:

	IF fb_state_entry.E THEN
		st_ctrl_out.b_fehler := fb_state_entry.i16_step = FEHLER;
		st_ctrl_out.b_gestoppt := fb_state_entry.i16_step = STOP;
		st_ctrl_out.b_busy:=FALSE;
		fb_ton_wz.IN:=TRUE;
	END_IF

	IF	fb_state_entry.fb_ton_Step.ET >t#5s THEN   (*Quittiert sich selbst*)
		fb_state_entry.i16_next_step:=INIT;
	END_IF

	IF fb_state_entry.X THEN
		fb_ton_wz.IN:=FALSE;
	END_IF

END_CASE
(*=======================================================*)
fb_state_entry(i16_pos:= 2);
st_ctrl_in:=st_ctrl_in_empty;

(* Fehlermeldungen und Betriebsmeldungen ab dem Startindex in die Meldungsarrays des fb_Fehlermeldung schreiben *)
garr_stoermeldungen[st_config.i16_meld_startindex +0] := b_sm[0];
garr_stoermeldungen[st_config.i16_meld_startindex +1] := b_sm[1];		(*Netzwerk nicht verbunden*)
garr_stoermeldungen[st_config.i16_meld_startindex +2] := b_sm[2];		(*User nicht vorhanden oder Passwort falsch*)
garr_stoermeldungen[st_config.i16_meld_startindex +3] := b_sm[3];		(*Verzeichnis nicht vorhanden!*)
garr_stoermeldungen[st_config.i16_meld_startindex +4] := b_sm[4];		(*Datei nicht vorhanden!*)
garr_stoermeldungen[st_config.i16_meld_startindex +5] := b_sm[5];
garr_stoermeldungen[st_config.i16_meld_startindex +6] := b_sm[6];
garr_stoermeldungen[st_config.i16_meld_startindex +7] := b_sm[7];
garr_stoermeldungen[st_config.i16_meld_startindex +8] := b_sm[8];
garr_stoermeldungen[st_config.i16_meld_startindex +9] := b_sm[9];
garr_stoermeldungen[st_config.i16_meld_startindex +10] := sm_DateiNichtVorhanden;
garr_stoermeldungen[st_config.i16_meld_startindex +11] := sm_FehlerBeimOeffnenDerDatei;
garr_stoermeldungen[st_config.i16_meld_startindex +12] := sm_FehlerBeimAuslesenDerDatei;
garr_stoermeldungen[st_config.i16_meld_startindex +13] := sm_FehlerBeimSchliessenDerDatei;
garr_stoermeldungen[st_config.i16_meld_startindex +14] := sm_FehlerBeimLoeschenDerDatei;
garr_stoermeldungen[st_config.i16_meld_startindex +15] := sm_KeineImportdateiVorhanden;
garr_stoermeldungen[st_config.i16_meld_startindex +16] := sm_KeineErrIdGefunden;
garr_stoermeldungen[st_config.i16_meld_startindex +17] := FALSE;
garr_stoermeldungen[st_config.i16_meld_startindex +18] := FALSE;
garr_stoermeldungen[st_config.i16_meld_startindex +19] := FALSE;

garr_betriebsmeldungen[st_config.i16_meld_startindex + 0] := b_bm[0];		(*OK*)
garr_betriebsmeldungen[st_config.i16_meld_startindex + 1] := b_bm[1];		(*keinen Unterschied gefunden*)
garr_betriebsmeldungen[st_config.i16_meld_startindex + 2] := b_bm[2];
garr_betriebsmeldungen[st_config.i16_meld_startindex + 3] := b_bm[3];
garr_betriebsmeldungen[st_config.i16_meld_startindex + 4] := b_bm[4];
garr_betriebsmeldungen[st_config.i16_meld_startindex + 5] := b_bm[5];
garr_betriebsmeldungen[st_config.i16_meld_startindex + 6] := b_bm[6];
garr_betriebsmeldungen[st_config.i16_meld_startindex + 7] := b_bm[7];
garr_betriebsmeldungen[st_config.i16_meld_startindex + 8] := b_bm[8];
garr_betriebsmeldungen[st_config.i16_meld_startindex + 9] := b_bm[9];


CallPrg();
END_FUNCTION_BLOCK
ACTION CallPrg:
IF 	FIND(s_script,'.bat') > 0 THEN


	NT_StartProcess(
		NETID:='',
		PATHSTR		:='C:\Windows\System32\cmd.exe',
		DIRNAME		:=s_path,
		COMNDLINE	:=CONCAT('/C start /b ', s_script),
		START			:=,
		TMOUT			:=DEFAULT_ADS_TIMEOUT);

ELSE
	NT_StartProcess(
		NETID:='',
		PATHSTR	:='C:\Windows\System32\wscript.exe',
		DIRNAME	:=s_path,
		COMNDLINE	:=s_script,
		START		:=,
		TMOUT		:=DEFAULT_ADS_TIMEOUT);
END_IF

fbFileOpen(
	sNetId:='',
	sPathName:= ,
	nMode:=FOPEN_MODEREAD,
	ePath:=PATH_GENERIC,
	bExecute:= ,
	tTimeout:=T#1s,
	hFile=> hFile);

fbFileRead(
	sNetId:='' ,
	hFile:=hFile,
	pReadBuff:= ADR(FileString)  ,
	cbReadLen:=SIZEOF(FileString)  ,
	tTimeout:=t#2s );

fbFileClose(
	sNetId:='',
	hFile:=hFile,
	bExecute:= ,
	tTimeout:=t#1s);

fbFileDelete(
	sNetId:= ,
	sPathName:= , 
	ePath:= PATH_GENERIC,
	bExecute:= ,
	tTimeout:= t#1s );
END_ACTION

(* POU EPT Lib/Funktionsbausteine/ST_StateEntry, ST *)
FUNCTION_BLOCK ST_StateEntry
VAR
	arr_last_step_history	: ARRAY[0..31] OF STRING(110);
	i 					: INT := 0;
	last_pos 				: INT := 0;
	interner_step			: INT := 0;
	s_stepTime 			: STRING;
END_VAR
VAR_OUTPUT
	i16_last_step 			: enum_step_nr := INIT_OBJ;	(* Der Schritt vor diesem Schritt *)
	i16_step 				: enum_step_nr := INIT_OBJ;	(* Diese variable soll vom "case step of" verwendet werden *)
	E					: BOOL;					(* Aktiv bei betreten des Steps *)
	X					: BOOL;					(* Aktiv beim verlassen des Steps *)
	b_error 				: BOOL := FALSE;			(* Ablauf Pos 1,2,1,2,1,2,... nicht richtig *)
	fb_ton_Step			: TON;
END_VAR
VAR_INPUT
	i16_next_step 		: enum_step_nr := INIT_OBJ;	(* Nächster schritt *)
	i16_pos 				: INT;					(* Pos = 1: Aufruf vor dem Case step of ---  Pos = 2: Aufruf nach dem Case step of*)
	s_debugtext			: STRING(100);
END_VAR
VAR CONSTANT
	t_MaxStepTime		: TIME := T#60S;
END_VAR
(*stepTime ermitteln*)
fb_ton_Step(IN:= , PT:=t_MaxStepTime , Q=>  , ET=> );
IF	i16_step = i16_next_step THEN
	fb_ton_Step.IN:=TRUE;
END_IF

IF NOT b_error THEN
	CASE interner_step OF
		0:
			(* Mitten im Schritt drin *)
			X := FALSE;
			E := FALSE;


			(* Schritt wird verlassen *)
			IF i16_step <> i16_next_step AND i16_pos = 1 THEN
				subrDebugtext();
				interner_step := 10;
				X := TRUE;
				E := FALSE;
				fb_ton_Step.IN:=FALSE;
			END_IF

		10:
			(* Eintritt in neuen Schritt *)
			IF i16_pos = 1 THEN
				X := FALSE;
				E := TRUE;

				(* Schalte Schritt weiter *)
				i16_last_step := i16_step;
				i16_step := i16_next_step;
				(* Baue Statehistory *)

				IF  E THEN
					FOR i:= 31 TO 1 BY -1 DO
						arr_last_step_history[i] := arr_last_step_history[i-1];
					END_FOR
					arr_last_step_history[0] := '';
					s_stepTime:='';
					s_debugtext:='';
				END_IF

				interner_step := 0;

			END_IF
	END_CASE
END_IF

IF 	(fb_ton_Step.ET >= T#200ms AND arr_last_step_history[0] = '') OR	(* Am Anfang Debugtext schreiben, damit etwas drin steht *)
	(fb_ton_Step.Q AND s_stepTime <> '>1m') THEN	(* Debugtext schreiben, wenn t_MaxStepTime erreicht wird *)
	subrDebugtext();
END_IF

(* Prüfe Baustein *)
IF 	i16_pos = last_pos THEN
	b_error := TRUE;
END_IF

last_pos := i16_pos;
END_FUNCTION_BLOCK
ACTION subrDebugtext:
s_stepTime:=ET_TO_STRING(fb_ton_Step.ET);
IF 	fb_ton_Step.ET >= t_MaxStepTime THEN
	s_stepTime:=CONCAT('>',s_StepTime);
END_IF

(* history zusammenbauen aus StepNr, StepTime und debugtext*)
CASE i16_step OF
	INIT_OBJ :			arr_last_step_history[0]:='INIT_OBJ';
	INIT :				arr_last_step_history[0]:='INIT';
	BEREIT :				arr_last_step_history[0]:='BEREIT';
	FEHLER :			arr_last_step_history[0]:='FEHLER';
	STOP :				arr_last_step_history[0]:='STOP';
	STILLSTAND :		arr_last_step_history[0]:='STILLSTAND';
	HALT :				arr_last_step_history[0]:='HALT';
	HANDRAD :			arr_last_step_history[0]:='HANDRAD';
	MOTORBREMSE_AUF :	arr_last_step_history[0]:='MOTORBREMSE_AUF';
	MOTORBREMSE_ZU :	arr_last_step_history[0]:='MOTORBREMSE_ZU';
	LUEFTEN :			arr_last_step_history[0]:='LUEFTEN';
	REGELN :			arr_last_step_history[0]:='REGELN';
	INBETRIEBNAHME :		arr_last_step_history[0]:='INBETRIEBNAHME';
	(* Zylinder *)
	ZYL_INIT :			arr_last_step_history[0]:='ZYL_INIT';
	GESTOPPT :			arr_last_step_history[0]:='GESTOPPT';
	EINGEFAHREN :		arr_last_step_history[0]:='EINGEFAHREN';
	BEWEGUNG_AUSFAHREN :		arr_last_step_history[0]:='BEWEGUNG_AUSFAHREN';
	AUSGEFAHREN :		arr_last_step_history[0]:='AUSGEFAHREN';
	BEWEGUNG_EINFAHREN :		arr_last_step_history[0]:='BEWEGUNG_EINFAHREN';
	MITTEGEFAHREN :		arr_last_step_history[0]:='MITTEGEFAHREN';
	BEWEGUNG_MITTE  :	arr_last_step_history[0]:='BEWEGUNG_MITTE';
	LUFTLOS :			arr_last_step_history[0]:='LUFTLOS';
	ZYL_FEHLER :		arr_last_step_history[0]:='ZYL_FEHLER';
	DIREKT_EINFAHREN :	arr_last_step_history[0]:='DIREKT_EINFAHREN';
	DIREKT_AUSFAHREN :	arr_last_step_history[0]:='DIREKT_AUSFAHREN';
ELSE
	arr_last_step_history[0] := INT_TO_STRING(i16_step);
END_CASE

IF 	s_stepTime ='0ms' OR s_stepTime =''THEN
	s_stepTime:='3ms';		(*damit nicht 0 drin steht*)
END_IF
arr_last_step_history[0] := CONCAT(arr_last_step_history[0],':  ');
arr_last_step_history[0] := CONCAT(arr_last_step_history[0],s_stepTime);
arr_last_step_history[0] := CONCAT(arr_last_step_history[0],': ');
arr_last_step_history[0] := CONCAT(arr_last_step_history[0],s_debugtext);
END_ACTION

(* POU EPT Lib/Funktionen/ET_TO_STRING, ST *)
FUNCTION ET_TO_STRING :STRING
VAR_INPUT
	et		:TIME;
END_VAR

VAR
	i16_LEN	:INT;
END_VAR
ET_TO_STRING:=TIME_TO_STRING(et);
ET_TO_STRING:=DELETE(ET_TO_STRING,2,1);

IF 	et> t#60s THEN
	ET_TO_STRING:=LEFT(ET_TO_STRING,FIND(ET_TO_STRING,'s'));
END_IF
END_FUNCTION

(* POU EPT Lib/Daten/ST_SaveAndLoad, ST *)
PROGRAM ST_SaveAndLoad
VAR_INPUT
	st_ctrl_in			: struct_ctrl_in;
	st_config			: struct_config;

END_VAR
VAR_OUTPUT
	st_ctrl_out			:struct_ctrl_out;
END_VAR
VAR
	b_init				:BOOL;
	fb_state_entry		:ST_StateEntry;
	fb_ton_quitt			:TON;

	NT_StartProcess 	: NT_StartProcess;
	fbFileDelete			: FB_FileDelete;

	s_script				: STRING;
	sm_FehlerBeimStartenDerBat				:BOOL;
	sm_FehlerBeimLoeschenDerDatei		:BOOL;

END_VAR
VAR CONSTANT
		s_bbgenMachineToSrv				:STRING:=		'_bbgen_aktuelles_wz_und_band_von_zelle_nach_server.bat';

		s_bbgenSrvToMachine				:STRING:=		'_bbgen_von_server_nach_zelle.bat';
		s_bbgenSrvToMachineHalbauto		:STRING:=		'_bbgen_von_server_nach_zelle_halbauto.bat';
		s_bbgenSrvToMachineManuell		:STRING:=		'_bbgen_von_server_nach_zelle_manuell.bat';

		s_fbwf_info							:STRING:=		'fbwf_info.bat';
		s_fbwf_disable						:STRING:=		'fbwf_disable.bat';
		s_fbwf_enable						:STRING:=		'fbwf_enable.bat';
END_VAR
(*======================================================
   ST_SaveAndLoad
 ------------------------------------------------------
   Auth: 		Werner Friedl   						 
   Date: 		06.10.2020   						     
   Rev.: 		1.0	
   Desc:		Die bat Datein zum laden und speichern der BBgen Dateien werden hier ausgeführt.
			mit der Constante b_wkzBereinigen kann bestimmt werden, ob die Werkzeugdateu forher gelöscht wird.

 ========================================================*)
IF	NOT b_init THEN
	b_Init:=TRUE;
END_IF
CallPrg();
(* ========================================================*)
fb_ton_quitt(IN:= , PT:= t#100ms, Q=> , ET=> );



fb_state_entry(i16_pos:= 1);
CASE fb_state_entry.i16_step OF
(*=======================================================*)
INIT_OBJ:
		fb_state_entry.i16_next_step := INIT;

(*=======================================================*)
INIT:
	IF	fb_state_entry.E THEN
		sm_FehlerBeimStartenDerBat:=FALSE;
		sm_FehlerBeimLoeschenDerDatei:=FALSE;
	END_IF

		fb_state_entry.i16_next_step := BEREIT;


(*=======================================================*)
BEREIT:	fb_state_entry.s_debugtext:='warte auf Taster Save oder Load';

	IF fb_state_entry.E THEN
		st_ctrl_out.b_bereit:=TRUE;
		NT_StartProcess.START:=FALSE;
	END_IF

	(*-----------------------Weiterschaltbedingungen----------------------------*)
	IF 	visu.b_load THEN
		fb_state_entry.i16_next_step:=110;
	ELSIF
		visu.b_save THEN
		IF 	gst_datensatz.st_md.b_wkzBereinigen THEN
			fb_state_entry.i16_next_step:=210;
		ELSE
			fb_state_entry.i16_next_step:=240;
		END_IF
	ELSIF
		visu.b_fbwf_info THEN
		s_script:=s_fbwf_info;
		fb_state_entry.i16_next_step:=120;
	ELSIF
		visu.b_fbwf_disable THEN
		s_script:=s_fbwf_disable;
		fb_state_entry.i16_next_step:=120;
	ELSIF
		visu.b_fbwf_enable THEN
		s_script:=s_fbwf_enable;
		fb_state_entry.i16_next_step:=120;
	END_IF

	IF fb_state_entry.X THEN
		st_ctrl_out.b_busy:=TRUE;
		st_ctrl_out.b_bereit := FALSE;
		st_ctrl_out.b_fertig := FALSE;
	END_IF

(*=======================================================*)
110:fb_state_entry.s_debugtext:='erstelle s_script';

	IF fb_state_entry.E THEN

 		CASE gst_datensatz.st_md.i16_typ_bestueckmodus OF

			BESTUECKUNG_MANUAL:
				s_script:=CONCAT(visu.s_akt_sprache,s_bbgenSrvToMachineManuell);

			BESTUECKUNG_HALBAUTO:
				s_script:=CONCAT(visu.s_akt_sprache,s_bbgenSrvToMachineHalbauto);

			BESTUECKUNG_AUTO:
				s_script:=CONCAT(visu.s_akt_sprache,s_bbgenSrvToMachine);
		END_CASE

		fb_state_entry.i16_next_step:=120;
	END_IF

(*=======================================================*)
120:fb_state_entry.s_debugtext:='start bat Script "Laden der Dateien vom Server"';

	IF 	fb_state_entry.E THEN
		NT_StartProcess.START:=TRUE;
	END_IF

	(*-----------------------Weiterschaltbedingungen----------------------------*)
	IF 	NT_StartProcess.BUSY THEN
		fb_state_entry.i16_next_step:=130;
	END_IF

	IF 	fb_state_entry.X THEN
		NT_StartProcess.START:=FALSE;
	END_IF

(*=======================================================*)
130:fb_state_entry.s_debugtext:='Warten auf fertig';

	IF 	NT_StartProcess.ERR THEN
		fb_state_entry.s_debugtext:=CONCAT(fb_state_entry.s_debugtext,' ERRID => ');
		fb_state_entry.s_debugtext:=CONCAT(fb_state_entry.s_debugtext,UDINT_TO_STRING(NT_StartProcess.ERRID));
		sm_FehlerBeimStartenDerBat:=TRUE;
		fb_state_entry.i16_next_step:=FEHLER;
	ELSIF
		NOT NT_StartProcess.BUSY AND
		NOT NT_StartProcess.ERR AND
		fb_state_entry.fb_ton_Step.ET>t#3000ms THEN
		st_ctrl_out.b_busy:=FALSE;
		st_ctrl_out.b_fertig := TRUE;
		fb_state_entry.i16_next_step:=BEREIT;
	END_IF

	IF 	fb_state_entry.X THEN
		visu.b_fbwf_info:=FALSE;
		visu.b_fbwf_disable:=FALSE;
		visu.b_fbwf_enable:=FALSE;
		visu.b_load:=FALSE;
	END_IF

(*=======================================================*)
(*=======================================================*)
210:	fb_state_entry.s_debugtext:='Löschen der Werkzeug Datei';

	IF 	fb_state_entry.E THEN
		fbFileDelete.sPathName:=CONCAT(CONCAT(ST_BBGen.s_wkz_path,gst_datensatz.st_md.s_aktuelles_wkz),'.xml');
		fbFileDelete.bExecute:=TRUE;
	END_IF

	(*-----------------------Weiterschaltbedingungen----------------------------*)
	IF 	fbFileDelete.bBusy THEN
		fb_state_entry.i16_next_step:=220;
	END_IF

	IF 	fb_state_entry.X THEN
		fbFileDelete.bExecute:=FALSE;
	END_IF

(*=======================================================*)
220: fb_state_entry.s_debugtext:='warte auf fertig';

	IF 	NOT fbFileDelete.bBusy THEN
		IF 	fbFileDelete.bError THEN
			fb_state_entry.s_debugtext:=CONCAT(fb_state_entry.s_debugtext,' ERRID => ');
			fb_state_entry.s_debugtext:=CONCAT(fb_state_entry.s_debugtext,UDINT_TO_STRING(fbFileDelete.nErrId));
			fb_state_entry.i16_next_step:=FEHLER;
			sm_FehlerBeimLoeschenDerDatei:=TRUE;
		ELSE
			fb_state_entry.i16_next_step:=230;
		END_IF
	END_IF

(*=======================================================*)
230: fb_state_entry.s_debugtext:='Werkzeugdatei neu erstellen';

	IF 	fb_state_entry.E THEN
		gi16_bbgen_auftrag:=SCHREIBE_WKZ;
	END_IF

	(*-----------------------Weiterschaltbedingungen----------------------------*)
	IF 	gi16_bbgen_auftrag = KEIN_BB_AUFTRAG THEN
		fb_state_entry.i16_next_step:=240;
	END_IF

(*=======================================================*)
240:	fb_state_entry.s_debugtext:='Speichern auf Server';

	IF 	fb_state_entry.E THEN
		s_script:=CONCAT(visu.s_akt_sprache,s_bbgenMachineToSrv);
		NT_StartProcess.START:=TRUE;
	END_IF

	(*-----------------------Weiterschaltbedingungen----------------------------*)
	IF 	NT_StartProcess.BUSY THEN
		fb_state_entry.i16_next_step:=250;
	END_IF

	IF 	fb_state_entry.X THEN
		NT_StartProcess.START:=FALSE;
	END_IF

(*=======================================================*)
250:fb_state_entry.s_debugtext:='Warten auf fertig';

	IF 	NT_StartProcess.ERR THEN
		fb_state_entry.s_debugtext:=CONCAT(fb_state_entry.s_debugtext,' ERRID => ');
		fb_state_entry.s_debugtext:=CONCAT(fb_state_entry.s_debugtext,UDINT_TO_STRING(NT_StartProcess.ERRID));
		sm_FehlerBeimStartenDerBat:=TRUE;
		fb_state_entry.i16_next_step:=FEHLER;
	ELSIF
		NOT NT_StartProcess.BUSY AND
		NOT NT_StartProcess.ERR AND
		fb_state_entry.fb_ton_Step.ET>t#3000ms THEN
		st_ctrl_out.b_busy:=FALSE;
		st_ctrl_out.b_fertig := TRUE;
		fb_state_entry.i16_next_step:=BEREIT;
	END_IF

	IF 	fb_state_entry.X THEN
		visu.b_save:=FALSE;
	END_IF

(*=======================================================*)
STOP, FEHLER:

	IF fb_state_entry.E THEN
		st_ctrl_out.b_fehler := fb_state_entry.i16_step = FEHLER;
		st_ctrl_out.b_gestoppt := fb_state_entry.i16_step = STOP;
		st_ctrl_out.b_busy:=FALSE;
	END_IF

	IF	fb_state_entry.fb_ton_Step.ET > t#1000ms THEN   (*Quittiert sich selbst*)
		fb_state_entry.i16_next_step:=INIT;
	END_IF

END_CASE

fb_state_entry(i16_pos:= 2 );
st_ctrl_in:=st_ctrl_in_empty;


garr_stoermeldungen[st_config.i16_meld_startindex + 0] := sm_FehlerBeimStartenDerBat;
garr_stoermeldungen[st_config.i16_meld_startindex + 1] := sm_FehlerBeimLoeschenDerDatei;
garr_stoermeldungen[st_config.i16_meld_startindex + 2] := FALSE;
garr_stoermeldungen[st_config.i16_meld_startindex + 3] := FALSE;
garr_stoermeldungen[st_config.i16_meld_startindex + 4] := FALSE;
garr_stoermeldungen[st_config.i16_meld_startindex + 5] := FALSE;
garr_stoermeldungen[st_config.i16_meld_startindex + 6] := FALSE;
garr_stoermeldungen[st_config.i16_meld_startindex + 7] := FALSE;
garr_stoermeldungen[st_config.i16_meld_startindex + 8] := FALSE;
garr_stoermeldungen[st_config.i16_meld_startindex + 9] := FALSE;
garr_stoermeldungen[st_config.i16_meld_startindex + 10] := FALSE;
garr_stoermeldungen[st_config.i16_meld_startindex + 11] := FALSE;
garr_stoermeldungen[st_config.i16_meld_startindex + 12] := FALSE;
garr_stoermeldungen[st_config.i16_meld_startindex + 13] := FALSE;
garr_stoermeldungen[st_config.i16_meld_startindex + 14] := FALSE;
garr_stoermeldungen[st_config.i16_meld_startindex + 15] := FALSE;
garr_stoermeldungen[st_config.i16_meld_startindex + 16] := FALSE;
garr_stoermeldungen[st_config.i16_meld_startindex + 17] := FALSE;
garr_stoermeldungen[st_config.i16_meld_startindex + 18] := FALSE;
garr_stoermeldungen[st_config.i16_meld_startindex + 19] := FALSE;

garr_betriebsmeldungen[st_config.i16_meld_startindex + 0] := FALSE;
garr_betriebsmeldungen[st_config.i16_meld_startindex + 1] := FALSE;
garr_betriebsmeldungen[st_config.i16_meld_startindex + 2] := FALSE;
garr_betriebsmeldungen[st_config.i16_meld_startindex + 3] := FALSE;
garr_betriebsmeldungen[st_config.i16_meld_startindex + 4] := FALSE;
garr_betriebsmeldungen[st_config.i16_meld_startindex + 5] := FALSE;
garr_betriebsmeldungen[st_config.i16_meld_startindex + 6] := FALSE;
garr_betriebsmeldungen[st_config.i16_meld_startindex + 7] := FALSE;
garr_betriebsmeldungen[st_config.i16_meld_startindex + 8] := FALSE;
garr_betriebsmeldungen[st_config.i16_meld_startindex + 9] := FALSE;
garr_betriebsmeldungen[st_config.i16_meld_startindex + 10] := FALSE;
garr_betriebsmeldungen[st_config.i16_meld_startindex + 11] := FALSE;
garr_betriebsmeldungen[st_config.i16_meld_startindex + 12] := FALSE;
garr_betriebsmeldungen[st_config.i16_meld_startindex + 13] := FALSE;
garr_betriebsmeldungen[st_config.i16_meld_startindex + 14] := FALSE;
garr_betriebsmeldungen[st_config.i16_meld_startindex + 15] := FALSE;
garr_betriebsmeldungen[st_config.i16_meld_startindex + 16] := FALSE;
garr_betriebsmeldungen[st_config.i16_meld_startindex + 17] := FALSE;
garr_betriebsmeldungen[st_config.i16_meld_startindex + 18] := FALSE;
garr_betriebsmeldungen[st_config.i16_meld_startindex + 19] := FALSE;
END_PROGRAM
ACTION CallPrg:
NT_StartProcess(
	NETID:='',
	PATHSTR		:='C:\Windows\System32\cmd.exe',
	DIRNAME		:=s_tools_path,
	COMNDLINE	:=CONCAT('/C start /b ', s_script),
	START			:=,
	TMOUT			:=DEFAULT_ADS_TIMEOUT);


fbFileDelete(
	sNetId:= ,
	sPathName:= , 
	ePath:= PATH_GENERIC,
	bExecute:= ,
	tTimeout:= t#1s );
END_ACTION

(* POU Gemeinsamkeiten17xx/BBGen/ST_BBGen, ST *)
PROGRAM ST_BBGen
VAR_INPUT
	st_config							: struct_config;
	st_ctrl_in							: struct_ctrl_in;
END_VAR
VAR_IN_OUT
	st_visu								: struct_xml_visu;
	i16_auftrag						: enum_bbgen_auftrag;
END_VAR
VAR_OUTPUT
	st_ctrl_out						: struct_ctrl_out;
END_VAR
VAR
	fb_state_entry						: ST_StateEntry;
	fb_state_entry2					: ST_StateEntry;
	fb_ton_quitt						: TON;
	fb_bbgen_xml_file					: ST_BBGenXMLFile;
	fb_bbgen_write_file				: ST_BBGenWriteFile;
	fb_wkz_band_wt_schreiben			: ST_Export_String;
	s_name_alt_wkz					: STRING;
	s_name_alt_band					: STRING;
	s_name_alt_wt					: STRING;
	fb_xml_srv_read					: FB_XmlSrvReadByName;
	s_PLC_path_name				: STRING(255);
	nErrId							: UDINT;

	(* Pfadnamen für die einzelnen Maschinendaten *)
	s_wkz_path						: STRING(50);
	s_isk_path						: STRING(50);
	s_bestueckbild_path				: STRING(50);
	s_bestueckbild_halbauto_path	: STRING(50);
	s_band_path					: STRING(50);
	s_wt_path						: STRING(50);

	(* BBGen: Step 520 *)
	st_akt_bestueckprogramm			: struct_bestueckprogramm;
	b_ok							: ARRAY[0..4] OF BOOL;
	b_sort_swap						: BOOL;
	tmp_y							: LREAL;
	tmp_z							: LREAL;
	tmp_b							: INT;
	swap_a							: DINT;
	swap_b							: DINT;

	s_md_name						: STRING(50);
	s_md_backup_name				: STRING(50);
	s_bestueckbild_name				: STRING(50);

	(* Temporäre Variable *)
	i								: DINT := 0;
	k								: DINT := 0;
	lr_tmp							: LREAL := 0.0;
	i16_tmp							: INT;
	i32_tmp							: DINT;
	hm_alle_daten_laden				: BOOL := FALSE;
	hm_alle_daten_speichern			: BOOL := FALSE;
	fb_r_trig_taste_wkz_laden			: R_TRIG;
	fb_r_trig_taste_wkz_speichern		: R_TRIG;
	b_first_cycle 						: BOOL := TRUE;
	fb_f_trig_steuerung				: F_TRIG;

	sm_fehler_lesen_wkz				: BOOL;
	sm_fehler_lesen_md				: BOOL;
	sm_fehler_lesen_isk				: BOOL;
	sm_fehler_lesen_band				: BOOL;
	sm_fehler_lesen_bestueckbild		: BOOL;
	sm_fehler_lesen_wt				: BOOL;
	sm_fehler_schreiben_wkz			: BOOL;
	sm_fehler_schreiben_md			: BOOL;
	sm_fehler_schreiben_isk			: BOOL;
	sm_fehler_schreiben_band			: BOOL;
	sm_fehler_schreiben_wt			: BOOL;
	sm_fehler_schreiben_bestueckbild	: BOOL;
	sm_fehler_generieren_bestueckbild	: BOOL;
	sm_fehler_schreiben_bestueckbild_auf_hdd : BOOL;
	sm_fehler_wkz_nicht_vorhanden		: BOOL;
	sm_fehler_falsches_Band			: BOOL;

	bm_kleinster_greifer_groesser_kleinste_pinanzahl_in_bb : BOOL;
	bm_keine_vollbestueck_Artikelnummer : BOOL;

	gst_datensatz_copy				: struct_datensatz;
	b_lesen_komplett					: BOOL:=FALSE;
	j								: INT:=0;
	hm_md_speichern					: BOOL;
	fb_r_trig_taste_bestueckprg_manuell	: R_TRIG;
	fb_ton_end						: TON;
	fb_ton_wz						: TON;

	(*Aktion: Hub_Faktor_ermitteln*)
	s_HelpBand						: ARRAY [0..14] OF STRING(50);
	i32_maxAnzahl					: DINT;
	i32_Anzahl						: ARRAY [0..14] OF DINT;
	m								: DINT;
	n								: DINT;
	lr_min_FaktorHub					: LREAL;
	lr_FaktorHub						: LREAL:=1;
	i32_UsedTool					: DINT := 0;
	fb_r_trig_taste_vollbestuecken		: R_TRIG;

	wkz_Nr							: INT:=-1;
	gst_manuelles_bestueckprogramm_copy	: struct_bestueckprogramm;

	(*wkz_gruppe*) (*nur bei Halbautomatisch: Werkzeuge die mann zusammenfassen kann*)

	st_wkz_gruppe_copy				: ARRAY[0..4] OF  struct_md_wkz;
	i32_neues_Wkz					: DINT;
	state							: INT;
	sm_Wkz_nicht_kompatibel			: BOOL;
	sm_Band_nicht_kompatibel			: BOOL;
	sm_Wkz_Gruppe_nicht_zugeordnet	: BOOL;
	b_Wkz_Gruppe_gebildet			: BOOL;
	i16_anzahl_Wkz_Gruppen			: INT;
	b_Wkz_akt_vorhanden				: BOOL;
	for_begin						: DINT;
	for_end							: DINT;
	st_wkz_leer						: struct_wkz;
	st_band_leer						: struct_banddaten;
	st_wt_leer						: struct_wt;
	st_bestueckprogramm_leer			: struct_bestueckprogramm;
	st_bestueckbild_leer				: struct_bestueckbild;
	st_bestueckbild_halbauto_leer		: struct_bestueckbild_halbauto;
END_VAR
(* Flankenauswertung der Tasten an der Bedienoberfläche *)
fb_r_trig_taste_wkz_laden(CLK:= st_visu .b_taste_daten_laden, Q=> );
fb_r_trig_taste_wkz_speichern(CLK:= st_visu.b_taste_daten_speichern, Q=> );
fb_f_trig_steuerung(CLK:= ST_Safetyprogramm.se_steuerung_ein, Q=> );

fb_ton_quitt(IN:= , PT:= t#100ms, Q=> , ET=> );

IF fb_state_entry.i16_next_step > INIT AND fb_state_entry.i16_next_step < FEHLER THEN
	IF	 fb_bbgen_xml_file.bError THEN
		fb_state_entry.i16_next_step := FEHLER;
	END_IF

END_IF

subr_Wkz_Band_Wt_schreiben();

IF	b_lesen_komplett THEN
	wkz_gruppe_kompatibel();
ELSE
	st_wkz_gruppe_copy:=gst_datensatz.st_md.st_wkz_gruppe;
END_IF

(*mit einem bestimmten Werkzeug eine gaze Reihe bestücken*)
fb_r_trig_taste_vollbestuecken(CLK:=
						visu.b_vollbestuecken AND
						gi16_maschinenstatusinfo <> STATUS_MASCHINE_ARBEITET ,
									Q=> );

IF	fb_r_trig_taste_vollbestuecken.Q THEN
	IF	visu.b_merker_vollbestuecken THEN
		visu.b_merker_vollbestuecken:=FALSE;
	ELSE
		visu.b_merker_vollbestuecken:=TRUE;
	END_IF
END_IF

IF	visu.b_merker_vollbestuecken THEN
	gst_datensatz.st_md.b_wt_transport_aktiv:=FALSE;
END_IF

(* ======================================Schrittkette======================================== *)
fb_state_entry(i16_pos:= 1 );

auto_speichern_laden();

CASE fb_state_entry.i16_step OF
(*=======================================================*)
	0:	(* Init *)
		fb_ton_quitt.IN := FALSE;
		st_ctrl_out.b_bereit := FALSE;
		st_ctrl_out.b_fehler := FALSE;
		sm_fehler_lesen_wkz := FALSE;
		sm_fehler_lesen_md := FALSE;
		sm_fehler_lesen_isk := FALSE;
		sm_fehler_lesen_band	:= FALSE;
		sm_fehler_lesen_wt := FALSE;
		sm_fehler_lesen_bestueckbild := FALSE;
		sm_fehler_schreiben_wkz := FALSE;
		sm_fehler_schreiben_md := FALSE;
		sm_fehler_schreiben_isk := FALSE;
		sm_fehler_schreiben_band	:= FALSE;
		sm_fehler_schreiben_wt := FALSE;
		sm_fehler_schreiben_bestueckbild := FALSE;
		sm_fehler_generieren_bestueckbild := FALSE;
		sm_fehler_schreiben_bestueckbild_auf_hdd := FALSE;
		sm_fehler_wkz_nicht_vorhanden:=FALSE;
		sm_fehler_falsches_Band:=FALSE;
		sm_Wkz_nicht_kompatibel:=FALSE;
		sm_Wkz_Gruppe_nicht_zugeordnet:=FALSE;
		sm_Band_nicht_kompatibel:=FALSE;
		bm_keine_vollbestueck_Artikelnummer:=FALSE;

		fb_bbgen_xml_file.start_lesen_wkz := FALSE;
		fb_bbgen_xml_file.start_lesen_md := FALSE;
		fb_bbgen_xml_file.start_lesen_isk := FALSE;
		fb_bbgen_xml_file.start_lesen_band := FALSE;
		fb_bbgen_xml_file.start_lesen_bestueckbild := FALSE;
		fb_bbgen_xml_file.start_lesen_bestueckbild_halbauto := FALSE;
		fb_bbgen_xml_file.start_schreiben_wkz := FALSE;
		fb_bbgen_xml_file.start_schreiben_md := FALSE;
		fb_bbgen_xml_file.start_schreiben_isk := FALSE;
		fb_bbgen_xml_file.start_schreiben_band := FALSE;
		fb_bbgen_xml_file.start_schreiben_bestueckbild := FALSE;
		fb_bbgen_xml_file.start_schreiben_bestueckbild_halbauto := FALSE;
		fb_bbgen_xml_file.bQuit := FALSE;
		hm_alle_daten_laden := FALSE;
		hm_alle_daten_speichern := FALSE;
		i16_auftrag := KEIN_BB_AUFTRAG;

		s_wkz_path := 'D:/BBGen/Wkz/';
		s_isk_path := 'D:/BBGen/ISK/';
		s_bestueckbild_path := 'D:/BBGen/Bestueckbild/';
		s_bestueckbild_halbauto_path := 'D:/BBGen/BestueckbildHalbauto/';
		s_band_path := 'D:/BBGen/Band/';
		s_wt_path := 'D:/BBGen/Wt/';

		s_md_name := 'Maschinendaten';
		s_md_backup_name := 'Maschinendaten_Backup';
		s_bestueckbild_name := 'Artikelnummer_Bestueckbild';

		(*-----------------------Weiterschaltbedingungen----------------------------*)
		IF b_first_cycle THEN
			fb_state_entry.i16_next_step := 10;
		ELSE
			fb_state_entry.i16_next_step := 40;
		END_IF

(*=======================================================*)
	10:	(* PLC Projectpfad mit Projektnamen aus TPY auslesen Achtung!! Bootprojekt muss erstellt sein *)
		(* Unter Projekt >> Optionen >> TwinCAT >> Symbolbeschreibung aus Datei herunterladen muss gesetzt sein *)
		IF fb_state_entry.E THEN
			fb_xml_srv_read.sFilePath:= 'c:\TwinCAT\Boot\CurrentPlc_1.tpy';
			fb_xml_srv_read.sXPath := '/PlcProjectInfo/ProjectInfo/Path';
			fb_xml_srv_read.sSymName:= 'ST_BBGen.s_PLC_path_name';
			fb_xml_srv_read.bExecute:= TRUE;
		END_IF

		(*-----------------------Weiterschaltbedingungen----------------------------*)
		IF fb_xml_srv_read.bBusy THEN
			fb_xml_srv_read.bExecute:= FALSE;
			fb_state_entry.i16_next_step := 20;
		END_IF

(*=======================================================*)
	20:	(* Lesevorgang erfolgreich? *)
		IF NOT fb_xml_srv_read.bBusy THEN
			IF NOT fb_xml_srv_read.bError THEN
				fb_state_entry.i16_next_step := 40;
			ELSE	(* Fehler *)
				s_PLC_path_name := '!!! not found !!!';
				nErrId := fb_xml_srv_read.nErrId;
				fb_state_entry.i16_next_step := 40;
			END_IF
		END_IF

		(* PLC Name und Pfad trennen *)
		s_PLC_name := s_PLC_path_name;
		i := 0;
		FOR i := 1 TO 30 DO
			s_PLC_name := DELETE(s_PLC_name, FIND(s_PLC_name,'\'),1);
		END_FOR

		s_PLC_Path := s_PLC_path_name;
		s_PLC_Path := DELETE(s_PLC_Path, LEN(s_PLC_path)-FIND(s_PLC_path, s_PLC_name) + 1, FIND(s_PLC_path, s_PLC_name));
		s_Projekt_path := s_PLC_Path;
		s_Projekt_path := DELETE(s_Projekt_path, LEN(s_Projekt_path)-FIND(s_Projekt_path,'PLC\')+1,FIND(s_Projekt_path, 'PLC\'));

(*=======================================================*)
	40: (* Warte auf Auftrag *)
		IF fb_state_entry.E THEN
			st_ctrl_out.b_bereit := TRUE;
			IF b_first_cycle THEN
				path();
				(* Zuerst müssen die Maschinendaten geladen werden, damit Infos über aktuelles Wkz, Band, Isk, u.s.w. vorhanden sind. *)
				i16_auftrag := LESE_KOMPLETT;
				b_first_cycle := FALSE;
			END_IF
		END_IF

		(*-----------------------Weiterschaltbedingungen----------------------------*)
		IF i16_auftrag > KEIN_BB_AUFTRAG THEN
			fb_state_entry.i16_next_step := 50;

(*
			(* gg: fake that we can generate on the PC *)
			fb_state_entry.i16_next_step := 300;
			gst_datensatz.st_md.s_aktuelles_band := '154-20011';
			(* gst_datensatz.st_md.s_aktueller_isk := '154-4002'; muss vom artikel kommen *)
			gst_datensatz.st_md.s_aktuelle_artikelnummer := '154-50021_0';
			hm_alle_daten_laden := TRUE;
			gi16_maschinenstatusinfo := STATUS_MASCHINE_ARBEITET;
*)			
		END_IF

		IF fb_r_trig_taste_wkz_laden.Q THEN
			hm_alle_daten_laden := TRUE;
			b_lesen_komplett:=FALSE;
			i16_auftrag := LESE_WKZ;	(*sonst gehen Maschinenparameter die noch nicht gespeichert wurden verloren *)
		END_IF

		IF fb_r_trig_taste_wkz_speichern.Q OR fb_f_trig_steuerung.Q THEN
			fb_state_entry.i16_next_step := 820;
			hm_alle_daten_speichern := TRUE;
		END_IF

(*=======================================================*)
	50: (* Auftragsauswahl *)

		(*-----------------------Weiterschaltbedingungen----------------------------*)
		CASE i16_auftrag OF
			LESE_MD:
				fb_state_entry.i16_next_step := 100;

			LESE_WKZ:
				fb_state_entry.i16_next_step := 200;

			LESE_BAND:
				fb_state_entry.i16_next_step := 300;

			LESE_WT:
				fb_state_entry.i16_next_step := 350;

			LESE_BESTUECKBILD:
				fb_state_entry.i16_next_step := 400;

			LESE_ISK:
				fb_state_entry.i16_next_step := 600;

			LESE_KOMPLETT:
				hm_alle_daten_laden := TRUE;
				fb_state_entry.i16_next_step := 100;

			SCHREIBE_ISK:
				fb_state_entry.i16_next_step := 800;

			SCHREIBE_WKZ:
				fb_state_entry.i16_next_step := 820;

			SCHREIBE_BAND:
				fb_state_entry.i16_next_step := 840;

			SCHREIBE_WT:
				fb_state_entry.i16_next_step := 860;

			SCHREIBE_MD:
				fb_state_entry.i16_next_step := 880;

			SCHREIBE_BESTUECKBILD:
				fb_state_entry.i16_next_step := 880;

		END_CASE

(*============================Laden===========================*)
	100:	(* Maschinendaten *)
		IF fb_state_entry.E THEN
			fb_bbgen_xml_file.start_lesen_md:= TRUE;
			fb_bbgen_xml_file.s_path := s_md_path;
			fb_bbgen_xml_file.s_md:= s_md_name;
		END_IF

		(*-----------------------Weiterschaltbedingungen----------------------------*)
		IF fb_bbgen_xml_file.fertig_lesen  AND NOT fb_state_entry.E THEN
			fb_state_entry.i16_next_step := 110;
		ELSIF fb_bbgen_xml_file.bError THEN
			sm_fehler_lesen_md := TRUE;
			fb_state_entry.i16_next_step := FEHLER;
		END_IF

(*=======================================================*)
	110:
		IF fb_state_entry.E THEN
			fb_bbgen_xml_file.start_lesen_md := FALSE;
			gst_datensatz_copy.st_md:= gst_datensatz.st_md ;
		END_IF

		(*-----------------------Weiterschaltbedingungen----------------------------*)
		IF hm_alle_daten_laden THEN
			fb_state_entry.i16_next_step := 200;
		ELSE
			fb_state_entry.i16_next_step := 999;
		END_IF

(*=======================================================*)
	200: (* Wkz daten *)
		IF fb_state_entry.E THEN
			gst_datensatz.st_wkz:=st_wkz_leer;
		END_IF

		(*-----------------------Weiterschaltbedingungen----------------------------*)
		IF gst_datensatz.st_md.s_aktuelles_wkz <>'' THEN
			fb_state_entry.i16_next_step := 210;
		ELSIF hm_alle_daten_laden  THEN
				fb_state_entry.i16_next_step := 300;
			ELSE
				fb_state_entry.i16_next_step := 999;
		END_IF

	210:
		IF fb_state_entry.E  THEN
			fb_bbgen_xml_file.start_lesen_wkz := TRUE;
			fb_bbgen_xml_file.s_path := s_wkz_path;
			fb_bbgen_xml_file.s_wkz := gst_datensatz.st_md.s_aktuelles_wkz;
		END_IF

		(*-----------------------Weiterschaltbedingungen----------------------------*)
		IF fb_bbgen_xml_file.fertig_lesen  AND NOT fb_state_entry.E THEN
			fb_state_entry.i16_next_step := 220;
		ELSIF fb_bbgen_xml_file.bError THEN
			sm_fehler_lesen_wkz := TRUE;
			fb_state_entry.i16_next_step := FEHLER;
		END_IF

(*=======================================================*)
	220:
		IF fb_state_entry.E THEN
			gst_datensatz_copy.st_wkz:= gst_datensatz.st_wkz ;
			fb_bbgen_xml_file.start_lesen_wkz := FALSE;
		END_IF

		(*-----------------------Weiterschaltbedingungen----------------------------*)
		IF hm_alle_daten_laden THEN
			fb_state_entry.i16_next_step := 300;
		ELSE
			IF gst_datensatz_copy.st_md.s_aktuelles_wkz<>gst_datensatz.st_md.s_aktuelles_wkz THEN
				fb_state_entry.i16_next_step := 880;
			ELSE
				fb_state_entry.i16_next_step := 999;
			END_IF
		END_IF

(*=======================================================*)
	300:	(* Band Daten *)
		IF fb_state_entry.E THEN
			gst_datensatz.st_band:=st_band_leer;
		END_IF

		(*-----------------------Weiterschaltbedingungen----------------------------*)
		IF 	gst_datensatz.st_md.s_aktuelles_band <>'' THEN
			fb_state_entry.i16_next_step := 310;
		ELSIF 	hm_alle_daten_laden  THEN
				fb_state_entry.i16_next_step := 350;
			ELSE
				fb_state_entry.i16_next_step := 999;
		END_IF

	310:
		IF fb_state_entry.E THEN
			fb_bbgen_xml_file.start_lesen_band := TRUE;
			fb_bbgen_xml_file.s_path := s_band_path;
			fb_bbgen_xml_file.s_band := gst_datensatz.st_md.s_aktuelles_band;
		END_IF

